LIN {X 0,Y 481.419,Z 1220.363,A -85,B 0,C 180,E1 16137.855,E2 16137.855} C_VEL
LIN {X 0,Y 478.712,Z 1232.005,A -85,B 0,C 180,E1 16135.215,E2 16135.215} C_VEL
LIN {X 0,Y 476.64,Z 1241.797,A -85,B 0,C 180,E1 16132.7,E2 16132.7} C_VEL
LIN {X 0,Y 474.973,Z 1250.804,A -85,B 0,C 180,E1 16130.064,E2 16130.064} C_VEL
LIN {X 0,Y 473.553,Z 1260.287,A -85,B 0,C 180,E1 16126.81,E2 16126.81} C_VEL
LIN {X 0,Y 472.68,Z 1267.551,A -85,B 0,C 180,E1 16123.701,E2 16123.701} C_VEL
LIN {X 0,Y 472.253,Z 1272.478,A -85,B 0,C 180,E1 16121.105,E2 16121.105} C_VEL
LIN {X 0,Y 472.039,Z 1276.348,A -85,B 0,C 180,E1 16118.523,E2 16118.523} C_VEL
LIN {X 0,Y 471.949,Z 1279.075,A -85,B 0,C 180,E1 16116.077,E2 16116.077} C_VEL
LIN {X 0,Y 471.914,Z 1280.879,A -85,B 0,C 180,E1 16113.641,E2 16113.641} C_VEL
LIN {X 0,Y 471.887,Z 1281.781,A -85,B 0,C 180,E1 16111.211,E2 16111.211} C_VEL
LIN {X 0,Y 471.88,Z 1281.802,A -85,B 0,C 180,E1 16108.904,E2 16108.904} C_VEL
LIN {X 0,Y 471.914,Z 1280.943,A -85,B 0,C 180,E1 16106.474,E2 16106.474} C_VEL
LIN {X 0,Y 471.945,Z 1279.181,A -85,B 0,C 180,E1 16104.038,E2 16104.038} C_VEL
LIN {X 0,Y 472.038,Z 1276.338,A -85,B 0,C 180,E1 16101.47,E2 16101.47} C_VEL
LIN {X 0,Y 472.253,Z 1272.465,A -85,B 0,C 180,E1 16098.888,E2 16098.888} C_VEL
LIN {X 0,Y 472.681,Z 1267.536,A -85,B 0,C 180,E1 16096.292,E2 16096.292} C_VEL
LIN {X 0,Y 473.556,Z 1260.267,A -85,B 0,C 180,E1 16093.183,E2 16093.183} C_VEL
LIN {X 0,Y 474.976,Z 1250.78,A -85,B 0,C 180,E1 16089.929,E2 16089.929} C_VEL
LIN {X 0,Y 476.646,Z 1241.775,A -85,B 0,C 180,E1 16087.292,E2 16087.292} C_VEL
LIN {X 0,Y 478.72,Z 1231.982,A -85,B 0,C 180,E1 16084.778,E2 16084.778} C_VEL
LIN {X 0,Y 481.427,Z 1220.335,A -85,B 0,C 180,E1 16082.138,E2 16082.138} C_VEL
LIN {X 0,Y 485.675,Z 1203.701,A -85,B 0,C 180,E1 16078.883,E2 16078.883} C_VEL
LIN {X 0,Y 489.378,Z 1189.815,A -85,B 0,C 180,E1 16076.517,E2 16076.517} C_VEL
LIN {X 0,Y 493.33,Z 1175.667,A -85,B 0,C 180,E1 16074.366,E2 16074.366} C_VEL
LIN {X 0,Y 498.099,Z 1158.939,A -85,B 0,C 180,E1 16072.099,E2 16072.099} C_VEL
LIN {X 0,Y 504.095,Z 1137.823,A -85,B 0,C 180,E1 16069.613,E2 16069.613} C_VEL
LIN {X 0,Y 509.017,Z 1120.127,A -85,B 0,C 180,E1 16067.791,E2 16067.791} C_VEL
LIN {X 0,Y 513.599,Z 1103.252,A -85,B 0,C 180,E1 16066.243,E2 16066.243} C_VEL
LIN {X 0,Y 518.369,Z 1085.032,A -85,B 0,C 180,E1 16064.753,E2 16064.753} C_VEL
LIN {X 0,Y 523.838,Z 1063.175,A -85,B 0,C 180,E1 16063.183,E2 16063.183} C_VEL
LIN {X 0,Y 529.388,Z 1038.821,A -85,B 0,C 180,E1 16061.694,E2 16061.694} C_VEL
LIN {X 0,Y 533.582,Z 1018.565,A -85,B 0,C 180,E1 16060.628,E2 16060.628} C_VEL
LIN {X 0,Y 537.435,Z 998.235,A -85,B 0,C 180,E1 16059.707,E2 16059.707} C_VEL
LIN {X 0,Y 540.948,Z 977.497,A -85,B 0,C 180,E1 16058.905,E2 16058.905} C_VEL
LIN {X 0,Y 544.217,Z 955.344,A -85,B 0,C 180,E1 16058.189,E2 16058.189} C_VEL
LIN {X 0,Y 547.645,Z 926.74,A -85,B 0,C 180,E1 16057.465,E2 16057.465} C_VEL
LIN {X 0,Y 549.736,Z 902.182,A -85,B 0,C 180,E1 16057.006,E2 16057.006} C_VEL
LIN {X 0,Y 559.407,Z 699.055,A -85,B 0,C 180,E1 16053.926,E2 16053.926} C_VEL
LIN {X 0,Y 566.879,Z 547.842,A -85,B 0,C 180,E1 16051.622,E2 16051.622} C_VEL
LIN {X 0,Y 558.19,Z 534.324,A -85,B 0,C 180,E1 16049.808,E2 16049.808} C_VEL
LIN {X 0,Y 548.445,Z 519.702,A -85,B 0,C 180,E1 16047.586,E2 16047.586} C_VEL
LIN {X 0,Y 539.985,Z 507.974,A -85,B 0,C 180,E1 16045.471,E2 16045.471} C_VEL
LIN {X 0,Y 533.469,Z 499.045,A -85,B 0,C 180,E1 16043.677,E2 16043.677} C_VEL
LIN {X 0,Y 530.435,Z 495.224,A -85,B 0,C 180,E1 16042.791,E2 16042.791} C_VEL
LIN {X 0,Y 526.117,Z 489.958,A -85,B 0,C 180,E1 16041.46,E2 16041.46} C_VEL
LIN {X 0,Y 522.215,Z 485.091,A -85,B 0,C 180,E1 16040.16,E2 16040.16} C_VEL
LIN {X 0,Y 517.865,Z 480.177,A -85,B 0,C 180,E1 16038.606,E2 16038.606} C_VEL
LIN {X 0,Y 516.561,Z 478.461,A -85,B 0,C 180,E1 16038.1,E2 16038.1} C_VEL
LIN {X 0,Y 513.201,Z 475.014,A -85,B 0,C 180,E1 16036.76,E2 16036.76} C_VEL
LIN {X 0,Y 511.516,Z 472.461,A -85,B 0,C 180,E1 16035.999,E2 16035.999} C_VEL
LIN {X 0,Y 508.063,Z 469.299,A -85,B 0,C 180,E1 16034.416,E2 16034.416} C_VEL
LIN {X 0,Y 506.144,Z 466.136,A -85,B 0,C 180,E1 16033.364,E2 16033.364} C_VEL
LIN {X 0,Y 502.842,Z 463.782,A -85,B 0,C 180,E1 16031.528,E2 16031.528} C_VEL
LIN {X 0,Y 500.679,Z 459.895,A -85,B 0,C 180,E1 16029.948,E2 16029.948} C_VEL
LIN {X 0,Y 496.132,Z 456.529,A -85,B 0,C 180,E1 16025.9,E2 16025.9} C_VEL
LIN {X 0,Y 494.701,Z 452.911,A -85,B 0,C 180,E1 16023.244,E2 16023.244} C_VEL
LIN {X 0,Y 494.82,Z 453.072,A -85,B 0,C 180,E1 16016.292,E2 16016.292} C_VEL
LIN {X 0,Y 496.254,Z 456.64,A -85,B 0,C 180,E1 16013.754,E2 16013.754} C_VEL
LIN {X 0,Y 500.015,Z 459.457,A -85,B 0,C 180,E1 16010.33,E2 16010.33} C_VEL
LIN {X 0,Y 500.722,Z 459.956,A -85,B 0,C 180,E1 16009.821,E2 16009.821} C_VEL
LIN {X 0,Y 502.632,Z 463.514,A -85,B 0,C 180,E1 16008.409,E2 16008.409} C_VEL
LIN {X 0,Y 505.987,Z 466.072,A -85,B 0,C 180,E1 16006.515,E2 16006.515} C_VEL
LIN {X 0,Y 506.599,Z 466.831,A -85,B 0,C 180,E1 16006.183,E2 16006.183} C_VEL
LIN {X 0,Y 509.251,Z 470.688,A -85,B 0,C 180,E1 16004.804,E2 16004.804} C_VEL
LIN {X 0,Y 512.017,Z 473.051,A -85,B 0,C 180,E1 16003.58,E2 16003.58} C_VEL
LIN {X 0,Y 515.107,Z 477.209,A -85,B 0,C 180,E1 16002.256,E2 16002.256} C_VEL
LIN {X 0,Y 517.415,Z 479.37,A -85,B 0,C 180,E1 16001.377,E2 16001.377} C_VEL
LIN {X 0,Y 520.927,Z 483.776,A -85,B 0,C 180,E1 16000.08,E2 16000.08} C_VEL
LIN {X 0,Y 522.605,Z 485.625,A -85,B 0,C 180,E1 15999.505,E2 15999.505} C_VEL
LIN {X 0,Y 526.557,Z 490.305,A -85,B 0,C 180,E1 15998.208,E2 15998.208} C_VEL
LIN {X 0,Y 532.62,Z 497.875,A -85,B 0,C 180,E1 15996.371,E2 15996.371} C_VEL
LIN {X 0,Y 537.377,Z 503.877,A -85,B 0,C 180,E1 15995.045,E2 15995.045} C_VEL
LIN {X 0,Y 544.823,Z 513.332,A -85,B 0,C 180,E1 15993.132,E2 15993.132} C_VEL
LIN {X 0,Y 555.695,Z 527.944,A -85,B 0,C 180,E1 15990.608,E2 15990.608} C_VEL
LIN {X 0,Y 565.27,Z 542.364,A -85,B 0,C 180,E1 15988.575,E2 15988.575} C_VEL
LIN {X 0,Y 566.874,Z 545.239,A -85,B 0,C 180,E1 15988.242,E2 15988.242} C_VEL
LIN {X 0,Y 556.219,Z 762.388,A -85,B 0,C 180,E1 15984.941,E2 15984.941} C_VEL
LIN {X 0,Y 549.836,Z 895.617,A -85,B 0,C 180,E1 15982.918,E2 15982.918} C_VEL
LIN {X 0,Y 547.564,Z 922.141,A -85,B 0,C 180,E1 15982.412,E2 15982.412} C_VEL
LIN {X 0,Y 544.257,Z 949.115,A -85,B 0,C 180,E1 15981.705,E2 15981.705} C_VEL
LIN {X 0,Y 541.194,Z 970.006,A -85,B 0,C 180,E1 15981.021,E2 15981.021} C_VEL
LIN {X 0,Y 537.814,Z 990.083,A -85,B 0,C 180,E1 15980.241,E2 15980.241} C_VEL
LIN {X 0,Y 533.985,Z 1010.34,A -85,B 0,C 180,E1 15979.322,E2 15979.322} C_VEL
LIN {X 0,Y 529.443,Z 1032.223,A -85,B 0,C 180,E1 15978.164,E2 15978.164} C_VEL
LIN {X 0,Y 523.423,Z 1058.102,A -85,B 0,C 180,E1 15976.546,E2 15976.546} C_VEL
LIN {X 0,Y 518.432,Z 1077.945,A -85,B 0,C 180,E1 15975.098,E2 15975.098} C_VEL
LIN {X 0,Y 513.656,Z 1096.024,A -85,B 0,C 180,E1 15973.602,E2 15973.602} C_VEL
LIN {X 0,Y 508.746,Z 1113.935,A -85,B 0,C 180,E1 15971.933,E2 15971.933} C_VEL
LIN {X 0,Y 502.694,Z 1135.256,A -85,B 0,C 180,E1 15969.667,E2 15969.667} C_VEL
LIN {X 0,Y 499.787,Z 1145.411,A -85,B 0,C 180,E1 15968.454,E2 15968.454} C_VEL
LIN {X 0,Y 497.444,Z 1150.756,A -85,B 0,C 180,E1 15967.865,E2 15967.865} C_VEL
LIN {X 0,Y 488.416,Z 1164.255,A -85,B 0,C 180,E1 15966.475,E2 15966.475} C_VEL
LIN {X 0,Y 486.11,Z 1169.146,A -85,B 0,C 180,E1 15965.825,E2 15965.825} C_VEL
LIN {X 0,Y 481.158,Z 1186.125,A -85,B 0,C 180,E1 15963.126,E2 15963.126} C_VEL
LIN {X 0,Y 476.645,Z 1201.723,A -85,B 0,C 180,E1 15960.232,E2 15960.232} C_VEL
LIN {X 0,Y 473.56,Z 1213.335,A -85,B 0,C 180,E1 15957.786,E2 15957.786} C_VEL
LIN {X 0,Y 470.892,Z 1224.082,A -85,B 0,C 180,E1 15955.234,E2 15955.234} C_VEL
LIN {X 0,Y 468.337,Z 1235.729,A -85,B 0,C 180,E1 15952.074,E2 15952.074} C_VEL
LIN {X 0,Y 466.403,Z 1245.831,A -85,B 0,C 180,E1 15948.761,E2 15948.761} C_VEL
LIN {X 0,Y 465.348,Z 1252.735,A -85,B 0,C 180,E1 15946.095,E2 15946.095} C_VEL
LIN {X 0,Y 464.648,Z 1258.556,A -85,B 0,C 180,E1 15943.424,E2 15943.424} C_VEL
LIN {X 0,Y 464.225,Z 1263.433,A -85,B 0,C 180,E1 15940.678,E2 15940.678} C_VEL
LIN {X 0,Y 463.98,Z 1268,A -85,B 0,C 180,E1 15937.308,E2 15937.308} C_VEL
LIN {X 0,Y 463.917,Z 1270.577,A -85,B 0,C 180,E1 15934.206,E2 15934.206} C_VEL
LIN {X 0,Y 463.905,Z 1271.703,A -85,B 0,C 180,E1 15931.609,E2 15931.609} C_VEL
LIN {X 0,Y 463.872,Z 1271.834,A -85,B 0,C 180,E1 15929.016,E2 15929.016} C_VEL
LIN {X 0,Y 463.912,Z 1271.04,A -85,B 0,C 180,E1 15926.544,E2 15926.544} C_VEL
LIN {X 0,Y 463.95,Z 1269.227,A -85,B 0,C 180,E1 15923.942,E2 15923.942} C_VEL
LIN {X 0,Y 464.049,Z 1266.403,A -85,B 0,C 180,E1 15921.329,E2 15921.329} C_VEL
LIN {X 0,Y 464.286,Z 1262.364,A -85,B 0,C 180,E1 15918.576,E2 15918.576} C_VEL
LIN {X 0,Y 464.772,Z 1257.203,A -85,B 0,C 180,E1 15915.808,E2 15915.808} C_VEL
LIN {X 0,Y 465.874,Z 1249.153,A -85,B 0,C 180,E1 15912.354,E2 15912.354} C_VEL
LIN {X 0,Y 467.362,Z 1240.467,A -85,B 0,C 180,E1 15909.334,E2 15909.334} C_VEL
LIN {X 0,Y 469.114,Z 1231.79,A -85,B 0,C 180,E1 15906.73,E2 15906.73} C_VEL
LIN {X 0,Y 471.317,Z 1222.278,A -85,B 0,C 180,E1 15904.226,E2 15904.226} C_VEL
LIN {X 0,Y 474.554,Z 1209.618,A -85,B 0,C 180,E1 15901.294,E2 15901.294} C_VEL
LIN {X 0,Y 478.758,Z 1194.258,A -85,B 0,C 180,E1 15898.25,E2 15898.25} C_VEL
LIN {X 0,Y 482.501,Z 1181.259,A -85,B 0,C 180,E1 15895.983,E2 15895.983} C_VEL
LIN {X 0,Y 486.555,Z 1167.656,A -85,B 0,C 180,E1 15893.864,E2 15893.864} C_VEL
LIN {X 0,Y 491.218,Z 1152.193,A -85,B 0,C 180,E1 15891.711,E2 15891.711} C_VEL
LIN {X 0,Y 497.188,Z 1132.548,A -85,B 0,C 180,E1 15889.304,E2 15889.304} C_VEL
LIN {X 0,Y 502.899,Z 1113.013,A -85,B 0,C 180,E1 15887.242,E2 15887.242} C_VEL
LIN {X 0,Y 507.858,Z 1095.621,A -85,B 0,C 180,E1 15885.618,E2 15885.618} C_VEL
LIN {X 0,Y 512.717,Z 1077.884,A -85,B 0,C 180,E1 15884.145,E2 15884.145} C_VEL
LIN {X 0,Y 517.775,Z 1058.428,A -85,B 0,C 180,E1 15882.718,E2 15882.718} C_VEL
LIN {X 0,Y 523.999,Z 1032.581,A -85,B 0,C 180,E1 15881.093,E2 15881.093} C_VEL
LIN {X 0,Y 528.687,Z 1010.722,A -85,B 0,C 180,E1 15879.931,E2 15879.931} C_VEL
LIN {X 0,Y 532.643,Z 990.44,A -85,B 0,C 180,E1 15879.006,E2 15879.006} C_VEL
LIN {X 0,Y 536.242,Z 969.723,A -85,B 0,C 180,E1 15878.201,E2 15878.201} C_VEL
LIN {X 0,Y 539.707,Z 946.697,A -85,B 0,C 180,E1 15877.455,E2 15877.455} C_VEL
LIN {X 0,Y 543.153,Z 917.776,A -85,B 0,C 180,E1 15876.73,E2 15876.73} C_VEL
LIN {X 0,Y 545.156,Z 894.477,A -85,B 0,C 180,E1 15876.295,E2 15876.295} C_VEL
LIN {X 0,Y 555.378,Z 688.317,A -85,B 0,C 180,E1 15873.155,E2 15873.155} C_VEL
LIN {X 0,Y 562.529,Z 549.365,A -85,B 0,C 180,E1 15871.029,E2 15871.029} C_VEL
LIN {X 0,Y 552.764,Z 534.378,A -85,B 0,C 180,E1 15868.907,E2 15868.907} C_VEL
LIN {X 0,Y 541.403,Z 519.012,A -85,B 0,C 180,E1 15866.193,E2 15866.193} C_VEL
LIN {X 0,Y 532.717,Z 507.898,A -85,B 0,C 180,E1 15863.859,E2 15863.859} C_VEL
LIN {X 0,Y 528.301,Z 502.407,A -85,B 0,C 180,E1 15862.559,E2 15862.559} C_VEL
LIN {X 0,Y 524.158,Z 497.301,A -85,B 0,C 180,E1 15861.251,E2 15861.251} C_VEL
LIN {X 0,Y 519.573,Z 491.687,A -85,B 0,C 180,E1 15859.681,E2 15859.681} C_VEL
LIN {X 0,Y 515.874,Z 487.212,A -85,B 0,C 180,E1 15858.3,E2 15858.3} C_VEL
LIN {X 0,Y 514.503,Z 485.734,A -85,B 0,C 180,E1 15857.765,E2 15857.765} C_VEL
LIN {X 0,Y 511.154,Z 481.865,A -85,B 0,C 180,E1 15856.361,E2 15856.361} C_VEL
LIN {X 0,Y 509.976,Z 480.144,A -85,B 0,C 180,E1 15855.815,E2 15855.815} C_VEL
LIN {X 0,Y 506.51,Z 476.774,A -85,B 0,C 180,E1 15854.169,E2 15854.169} C_VEL
LIN {X 0,Y 504.733,Z 473.91,A -85,B 0,C 180,E1 15853.169,E2 15853.169} C_VEL
LIN {X 0,Y 501.451,Z 471.401,A -85,B 0,C 180,E1 15851.269,E2 15851.269} C_VEL
LIN {X 0,Y 499.227,Z 467.473,A -85,B 0,C 180,E1 15849.569,E2 15849.569} C_VEL
LIN {X 0,Y 495.28,Z 464.726,A -85,B 0,C 180,E1 15845.91,E2 15845.91} C_VEL
LIN {X 0,Y 493.731,Z 460.864,A -85,B 0,C 180,E1 15842.786,E2 15842.786} C_VEL
LIN {X 0,Y 493.807,Z 461.029,A -85,B 0,C 180,E1 15837.098,E2 15837.098} C_VEL
LIN {X 0,Y 495.742,Z 465.272,A -85,B 0,C 180,E1 15833.631,E2 15833.631} C_VEL
LIN {X 0,Y 499.508,Z 467.827,A -85,B 0,C 180,E1 15830.32,E2 15830.32} C_VEL
LIN {X 0,Y 501.609,Z 471.614,A -85,B 0,C 180,E1 15828.735,E2 15828.735} C_VEL
LIN {X 0,Y 505.115,Z 474.417,A -85,B 0,C 180,E1 15826.725,E2 15826.725} C_VEL
LIN {X 0,Y 508.144,Z 478.707,A -85,B 0,C 180,E1 15825.12,E2 15825.12} C_VEL
LIN {X 0,Y 510.497,Z 480.794,A -85,B 0,C 180,E1 15824.056,E2 15824.056} C_VEL
LIN {X 0,Y 513.661,Z 485.023,A -85,B 0,C 180,E1 15822.673,E2 15822.673} C_VEL
LIN {X 0,Y 515.722,Z 486.993,A -85,B 0,C 180,E1 15821.87,E2 15821.87} C_VEL
LIN {X 0,Y 519.4,Z 491.534,A -85,B 0,C 180,E1 15820.488,E2 15820.488} C_VEL
LIN {X 0,Y 521.036,Z 493.538,A -85,B 0,C 180,E1 15819.909,E2 15819.909} C_VEL
LIN {X 0,Y 525.9,Z 499.458,A -85,B 0,C 180,E1 15818.297,E2 15818.297} C_VEL
LIN {X 0,Y 530.608,Z 505.302,A -85,B 0,C 180,E1 15816.859,E2 15816.859} C_VEL
LIN {X 0,Y 536.955,Z 514.063,A -85,B 0,C 180,E1 15815.053,E2 15815.053} C_VEL
LIN {X 0,Y 543.856,Z 523.758,A -85,B 0,C 180,E1 15813.258,E2 15813.258} C_VEL
LIN {X 0,Y 552.297,Z 536.23,A -85,B 0,C 180,E1 15811.241,E2 15811.241} C_VEL
LIN {X 0,Y 562.019,Z 551.359,A -85,B 0,C 180,E1 15809.118,E2 15809.118} C_VEL
LIN {X 0,Y 562.519,Z 552.506,A -85,B 0,C 180,E1 15809.005,E2 15809.005} C_VEL
LIN {X 0,Y 551.538,Z 769.195,A -85,B 0,C 180,E1 15805.698,E2 15805.698} C_VEL
LIN {X 0,Y 544.926,Z 902.792,A -85,B 0,C 180,E1 15803.66,E2 15803.66} C_VEL
LIN {X 0,Y 542.526,Z 929.769,A -85,B 0,C 180,E1 15803.148,E2 15803.148} C_VEL
LIN {X 0,Y 539.082,Z 956.677,A -85,B 0,C 180,E1 15802.446,E2 15802.446} C_VEL
LIN {X 0,Y 535.875,Z 977.691,A -85,B 0,C 180,E1 15801.762,E2 15801.762} C_VEL
LIN {X 0,Y 532.498,Z 997.1,A -85,B 0,C 180,E1 15801.013,E2 15801.013} C_VEL
LIN {X 0,Y 528.51,Z 1017.543,A -85,B 0,C 180,E1 15800.092,E2 15800.092} C_VEL
LIN {X 0,Y 524.246,Z 1037.558,A -85,B 0,C 180,E1 15799.042,E2 15799.042} C_VEL
LIN {X 0,Y 518.513,Z 1062.103,A -85,B 0,C 180,E1 15797.551,E2 15797.551} C_VEL
LIN {X 0,Y 512.9,Z 1083.81,A -85,B 0,C 180,E1 15795.994,E2 15795.994} C_VEL
LIN {X 0,Y 508.189,Z 1101.184,A -85,B 0,C 180,E1 15794.581,E2 15794.581} C_VEL
LIN {X 0,Y 503.406,Z 1118.141,A -85,B 0,C 180,E1 15793.034,E2 15793.034} C_VEL
LIN {X 0,Y 498.461,Z 1135.191,A -85,B 0,C 180,E1 15791.29,E2 15791.29} C_VEL
LIN {X 0,Y 493.227,Z 1153.063,A -85,B 0,C 180,E1 15789.228,E2 15789.228} C_VEL
LIN {X 0,Y 487.168,Z 1173.445,A -85,B 0,C 180,E1 15786.521,E2 15786.521} C_VEL
LIN {X 0,Y 482.821,Z 1188.219,A -85,B 0,C 180,E1 15784.278,E2 15784.278} C_VEL
LIN {X 0,Y 479.025,Z 1201.533,A -85,B 0,C 180,E1 15782.012,E2 15782.012} C_VEL
LIN {X 0,Y 475.415,Z 1214.893,A -85,B 0,C 180,E1 15779.457,E2 15779.457} C_VEL
LIN {X 0,Y 471.628,Z 1229.839,A -85,B 0,C 180,E1 15776.161,E2 15776.161} C_VEL
LIN {X 0,Y 469.247,Z 1240.319,A -85,B 0,C 180,E1 15773.477,E2 15773.477} C_VEL
LIN {X 0,Y 467.508,Z 1249.081,A -85,B 0,C 180,E1 15770.922,E2 15770.922} C_VEL
LIN {X 0,Y 466.111,Z 1257.063,A -85,B 0,C 180,E1 15768.247,E2 15768.247} C_VEL
LIN {X 0,Y 465.127,Z 1264.171,A -85,B 0,C 180,E1 15765.455,E2 15765.455} C_VEL
LIN {X 0,Y 464.372,Z 1271.415,A -85,B 0,C 180,E1 15761.925,E2 15761.925} C_VEL
LIN {X 0,Y 464.051,Z 1275.866,A -85,B 0,C 180,E1 15759.046,E2 15759.046} C_VEL
LIN {X 0,Y 463.959,Z 1278.845,A -85,B 0,C 180,E1 15756.431,E2 15756.431} C_VEL
LIN {X 0,Y 463.916,Z 1280.743,A -85,B 0,C 180,E1 15753.951,E2 15753.951} C_VEL
LIN {X 0,Y 463.902,Z 1281.735,A -85,B 0,C 180,E1 15751.478,E2 15751.478} C_VEL
LIN {X 0,Y 463.875,Z 1281.824,A -85,B 0,C 180,E1 15749.008,E2 15749.008} C_VEL
LIN {X 0,Y 463.914,Z 1281.011,A -85,B 0,C 180,E1 15746.537,E2 15746.537} C_VEL
LIN {X 0,Y 463.949,Z 1279.178,A -85,B 0,C 180,E1 15743.935,E2 15743.935} C_VEL
LIN {X 0,Y 464.05,Z 1276.335,A -85,B 0,C 180,E1 15741.322,E2 15741.322} C_VEL
LIN {X 0,Y 464.265,Z 1272.654,A -85,B 0,C 180,E1 15738.82,E2 15738.82} C_VEL
LIN {X 0,Y 464.706,Z 1267.729,A -85,B 0,C 180,E1 15736.179,E2 15736.179} C_VEL
LIN {X 0,Y 465.528,Z 1261.094,A -85,B 0,C 180,E1 15733.27,E2 15733.27} C_VEL
LIN {X 0,Y 467.047,Z 1251.505,A -85,B 0,C 180,E1 15729.835,E2 15729.835} C_VEL
LIN {X 0,Y 468.861,Z 1242.145,A -85,B 0,C 180,E1 15727.026,E2 15727.026} C_VEL
LIN {X 0,Y 471.035,Z 1232.409,A -85,B 0,C 180,E1 15724.472,E2 15724.472} C_VEL
LIN {X 0,Y 473.711,Z 1221.398,A -85,B 0,C 180,E1 15721.918,E2 15721.918} C_VEL
LIN {X 0,Y 477.562,Z 1207.101,A -85,B 0,C 180,E1 15718.996,E2 15718.996} C_VEL
LIN {X 0,Y 481.936,Z 1191.272,A -85,B 0,C 180,E1 15716.216,E2 15716.216} C_VEL
LIN {X 0,Y 486.155,Z 1176.791,A -85,B 0,C 180,E1 15713.967,E2 15713.967} C_VEL
LIN {X 0,Y 490.64,Z 1161.636,A -85,B 0,C 180,E1 15711.865,E2 15711.865} C_VEL
LIN {X 0,Y 496.05,Z 1143.538,A -85,B 0,C 180,E1 15709.636,E2 15709.636} C_VEL
LIN {X 0,Y 502.349,Z 1121.865,A -85,B 0,C 180,E1 15707.331,E2 15707.331} C_VEL
LIN {X 0,Y 507.37,Z 1104.081,A -85,B 0,C 180,E1 15705.674,E2 15705.674} C_VEL
LIN {X 0,Y 512.117,Z 1086.627,A -85,B 0,C 180,E1 15704.228,E2 15704.228} C_VEL
LIN {X 0,Y 516.949,Z 1067.962,A -85,B 0,C 180,E1 15702.854,E2 15702.854} C_VEL
LIN {X 0,Y 522.724,Z 1044.339,A -85,B 0,C 180,E1 15701.339,E2 15701.339} C_VEL
LIN {X 0,Y 528.073,Z 1019.603,A -85,B 0,C 180,E1 15700.011,E2 15700.011} C_VEL
LIN {X 0,Y 532.037,Z 999.427,A -85,B 0,C 180,E1 15699.087,E2 15699.087} C_VEL
LIN {X 0,Y 535.649,Z 978.884,A -85,B 0,C 180,E1 15698.283,E2 15698.283} C_VEL
LIN {X 0,Y 538.892,Z 957.744,A -85,B 0,C 180,E1 15697.589,E2 15697.589} C_VEL
LIN {X 0,Y 542.016,Z 933.624,A -85,B 0,C 180,E1 15696.946,E2 15696.946} C_VEL
LIN {X 0,Y 544.766,Z 904.653,A -85,B 0,C 180,E1 15696.373,E2 15696.373} C_VEL
LIN {X 0,Y 548.192,Z 837.513,A -85,B 0,C 180,E1 15695.34,E2 15695.34} C_VEL
LIN {X 0,Y 558.918,Z 620.585,A -85,B 0,C 180,E1 15692.04,E2 15692.04} C_VEL
LIN {X 0,Y 562.397,Z 552.084,A -85,B 0,C 180,E1 15690.978,E2 15690.978} C_VEL
LIN {X 0,Y 553.476,Z 538.084,A -85,B 0,C 180,E1 15689.046,E2 15689.046} C_VEL
LIN {X 0,Y 544.949,Z 525.376,A -85,B 0,C 180,E1 15687.038,E2 15687.038} C_VEL
LIN {X 0,Y 537.505,Z 514.862,A -85,B 0,C 180,E1 15685.126,E2 15685.126} C_VEL
LIN {X 0,Y 530.745,Z 505.498,A -85,B 0,C 180,E1 15683.217,E2 15683.217} C_VEL
LIN {X 0,Y 527.928,Z 502.032,A -85,B 0,C 180,E1 15682.377,E2 15682.377} C_VEL
LIN {X 0,Y 524.176,Z 497.346,A -85,B 0,C 180,E1 15681.191,E2 15681.191} C_VEL
LIN {X 0,Y 519.572,Z 491.7,A -85,B 0,C 180,E1 15679.622,E2 15679.622} C_VEL
LIN {X 0,Y 515.853,Z 487.221,A -85,B 0,C 180,E1 15678.243,E2 15678.243} C_VEL
LIN {X 0,Y 514.617,Z 485.836,A -85,B 0,C 180,E1 15677.761,E2 15677.761} C_VEL
LIN {X 0,Y 511.231,Z 482.013,A -85,B 0,C 180,E1 15676.358,E2 15676.358} C_VEL
LIN {X 0,Y 510.053,Z 480.185,A -85,B 0,C 180,E1 15675.813,E2 15675.813} C_VEL
LIN {X 0,Y 506.544,Z 476.847,A -85,B 0,C 180,E1 15674.168,E2 15674.168} C_VEL
LIN {X 0,Y 504.751,Z 473.922,A -85,B 0,C 180,E1 15673.168,E2 15673.168} C_VEL
LIN {X 0,Y 501.431,Z 471.371,A -85,B 0,C 180,E1 15671.269,E2 15671.269} C_VEL
LIN {X 0,Y 499.167,Z 467.442,A -85,B 0,C 180,E1 15669.57,E2 15669.57} C_VEL
LIN {X 0,Y 495.337,Z 464.784,A -85,B 0,C 180,E1 15666.142,E2 15666.142} C_VEL
LIN {X 0,Y 493.671,Z 460.844,A -85,B 0,C 180,E1 15663.135,E2 15663.135} C_VEL
LIN {X 0,Y 493.79,Z 460.974,A -85,B 0,C 180,E1 15656.401,E2 15656.401} C_VEL
LIN {X 0,Y 495.186,Z 464.519,A -85,B 0,C 180,E1 15653.856,E2 15653.856} C_VEL
LIN {X 0,Y 498.894,Z 467.351,A -85,B 0,C 180,E1 15650.424,E2 15650.424} C_VEL
LIN {X 0,Y 499.505,Z 467.867,A -85,B 0,C 180,E1 15649.971,E2 15649.971} C_VEL
LIN {X 0,Y 501.483,Z 471.417,A -85,B 0,C 180,E1 15648.499,E2 15648.499} C_VEL
LIN {X 0,Y 505.11,Z 474.388,A -85,B 0,C 180,E1 15646.433,E2 15646.433} C_VEL
LIN {X 0,Y 507.821,Z 478.379,A -85,B 0,C 180,E1 15644.994,E2 15644.994} C_VEL
LIN {X 0,Y 510.484,Z 480.731,A -85,B 0,C 180,E1 15643.792,E2 15643.792} C_VEL
LIN {X 0,Y 513.739,Z 485.029,A -85,B 0,C 180,E1 15642.383,E2 15642.383} C_VEL
LIN {X 0,Y 515.742,Z 486.957,A -85,B 0,C 180,E1 15641.607,E2 15641.607} C_VEL
LIN {X 0,Y 519.364,Z 491.466,A -85,B 0,C 180,E1 15640.252,E2 15640.252} C_VEL
LIN {X 0,Y 521.084,Z 493.559,A -85,B 0,C 180,E1 15639.647,E2 15639.647} C_VEL
LIN {X 0,Y 525.893,Z 499.386,A -85,B 0,C 180,E1 15638.061,E2 15638.061} C_VEL
LIN {X 0,Y 530.597,Z 505.253,A -85,B 0,C 180,E1 15636.629,E2 15636.629} C_VEL
LIN {X 0,Y 535.39,Z 511.381,A -85,B 0,C 180,E1 15635.27,E2 15635.27} C_VEL
LIN {X 0,Y 542.663,Z 520.763,A -85,B 0,C 180,E1 15633.371,E2 15633.371} C_VEL
LIN {X 0,Y 553.115,Z 534.981,A -85,B 0,C 180,E1 15630.903,E2 15630.903} C_VEL
LIN {X 0,Y 562.472,Z 549.3,A -85,B 0,C 180,E1 15628.878,E2 15628.878} C_VEL
LIN {X 0,Y 551.643,Z 762.631,A -85,B 0,C 180,E1 15625.621,E2 15625.621} C_VEL
LIN {X 0,Y 545.038,Z 895.729,A -85,B 0,C 180,E1 15623.591,E2 15623.591} C_VEL
LIN {X 0,Y 542.693,Z 922.339,A -85,B 0,C 180,E1 15623.082,E2 15623.082} C_VEL
LIN {X 0,Y 539.287,Z 949.325,A -85,B 0,C 180,E1 15622.373,E2 15622.373} C_VEL
LIN {X 0,Y 536.026,Z 970.844,A -85,B 0,C 180,E1 15621.666,E2 15621.666} C_VEL
LIN {X 0,Y 532.442,Z 991.404,A -85,B 0,C 180,E1 15620.86,E2 15620.86} C_VEL
LIN {X 0,Y 528.266,Z 1012.692,A -85,B 0,C 180,E1 15619.88,E2 15619.88} C_VEL
LIN {X 0,Y 522.486,Z 1038.981,A -85,B 0,C 180,E1 15618.442,E2 15618.442} C_VEL
LIN {X 0,Y 517.18,Z 1060.623,A -85,B 0,C 180,E1 15617.037,E2 15617.037} C_VEL
LIN {X 0,Y 512.443,Z 1078.806,A -85,B 0,C 180,E1 15615.69,E2 15615.69} C_VEL
LIN {X 0,Y 507.598,Z 1096.478,A -85,B 0,C 180,E1 15614.215,E2 15614.215} C_VEL
LIN {X 0,Y 502.258,Z 1115.242,A -85,B 0,C 180,E1 15612.447,E2 15612.447} C_VEL
LIN {X 0,Y 495.703,Z 1137.269,A -85,B 0,C 180,E1 15610.052,E2 15610.052} C_VEL
LIN {X 0,Y 490.707,Z 1153.829,A -85,B 0,C 180,E1 15607.981,E2 15607.981} C_VEL
LIN {X 0,Y 486.216,Z 1168.784,A -85,B 0,C 180,E1 15605.879,E2 15605.879} C_VEL
LIN {X 0,Y 486.11,Z 1169.146,A -85,B 0,C 180,E1 15605.825,E2 15605.825} C_VEL
LIN {X 0,Y 483.843,Z 1174.1,A -85,B 0,C 180,E1 15605.162,E2 15605.162} C_VEL
LIN {X 0,Y 474.567,Z 1187.024,A -85,B 0,C 180,E1 15603.482,E2 15603.482} C_VEL
LIN {X 0,Y 472.731,Z 1190.74,A -85,B 0,C 180,E1 15602.858,E2 15602.858} C_VEL
LIN {X 0,Y 469.054,Z 1203.08,A -85,B 0,C 180,E1 15600.49,E2 15600.49} C_VEL
LIN {X 0,Y 465.9,Z 1214.435,A -85,B 0,C 180,E1 15598.037,E2 15598.037} C_VEL
LIN {X 0,Y 462.783,Z 1226.606,A -85,B 0,C 180,E1 15595.057,E2 15595.057} C_VEL
LIN {X 0,Y 460.106,Z 1238.252,A -85,B 0,C 180,E1 15591.684,E2 15591.684} C_VEL
LIN {X 0,Y 458.525,Z 1246.273,A -85,B 0,C 180,E1 15588.963,E2 15588.963} C_VEL
LIN {X 0,Y 457.415,Z 1253.127,A -85,B 0,C 180,E1 15586.251,E2 15586.251} C_VEL
LIN {X 0,Y 456.686,Z 1258.863,A -85,B 0,C 180,E1 15583.552,E2 15583.552} C_VEL
LIN {X 0,Y 456.223,Z 1263.932,A -85,B 0,C 180,E1 15580.612,E2 15580.612} C_VEL
LIN {X 0,Y 455.984,Z 1268.279,A -85,B 0,C 180,E1 15577.184,E2 15577.184} C_VEL
LIN {X 0,Y 455.917,Z 1270.672,A -85,B 0,C 180,E1 15574.154,E2 15574.154} C_VEL
LIN {X 0,Y 455.904,Z 1271.741,A -85,B 0,C 180,E1 15571.512,E2 15571.512} C_VEL
LIN {X 0,Y 455.873,Z 1271.848,A -85,B 0,C 180,E1 15568.998,E2 15568.998} C_VEL
LIN {X 0,Y 455.912,Z 1271.062,A -85,B 0,C 180,E1 15566.483,E2 15566.483} C_VEL
LIN {X 0,Y 455.953,Z 1269.266,A -85,B 0,C 180,E1 15563.835,E2 15563.835} C_VEL
LIN {X 0,Y 456.057,Z 1266.471,A -85,B 0,C 180,E1 15561.176,E2 15561.176} C_VEL
LIN {X 0,Y 456.304,Z 1262.656,A -85,B 0,C 180,E1 15558.502,E2 15558.502} C_VEL
LIN {X 0,Y 456.785,Z 1257.794,A -85,B 0,C 180,E1 15555.813,E2 15555.813} C_VEL
LIN {X 0,Y 457.759,Z 1250.951,A -85,B 0,C 180,E1 15552.723,E2 15552.723} C_VEL
LIN {X 0,Y 459.457,Z 1241.359,A -85,B 0,C 180,E1 15549.228,E2 15549.228} C_VEL
LIN {X 0,Y 461.371,Z 1232.339,A -85,B 0,C 180,E1 15546.454,E2 15546.454} C_VEL
LIN {X 0,Y 463.672,Z 1222.877,A -85,B 0,C 180,E1 15543.907,E2 15543.907} C_VEL
LIN {X 0,Y 466.722,Z 1211.414,A -85,B 0,C 180,E1 15541.187,E2 15541.187} C_VEL
LIN {X 0,Y 471.246,Z 1195.738,A -85,B 0,C 180,E1 15537.97,E2 15537.97} C_VEL
LIN {X 0,Y 475.577,Z 1181.347,A -85,B 0,C 180,E1 15535.418,E2 15535.418} C_VEL
LIN {X 0,Y 479.817,Z 1167.744,A -85,B 0,C 180,E1 15533.274,E2 15533.274} C_VEL
LIN {X 0,Y 484.702,Z 1152.233,A -85,B 0,C 180,E1 15531.093,E2 15531.093} C_VEL
LIN {X 0,Y 490.977,Z 1132.377,A -85,B 0,C 180,E1 15528.642,E2 15528.642} C_VEL
LIN {X 0,Y 496.805,Z 1113.177,A -85,B 0,C 180,E1 15526.599,E2 15526.599} C_VEL
LIN {X 0,Y 501.86,Z 1096.108,A -85,B 0,C 180,E1 15524.993,E2 15524.993} C_VEL
LIN {X 0,Y 506.92,Z 1078.302,A -85,B 0,C 180,E1 15523.504,E2 15523.504} C_VEL
LIN {X 0,Y 512.025,Z 1059.321,A -85,B 0,C 180,E1 15522.1,E2 15522.1} C_VEL
LIN {X 0,Y 518.219,Z 1034.667,A -85,B 0,C 180,E1 15520.525,E2 15520.525} C_VEL
LIN {X 0,Y 523.267,Z 1011.93,A -85,B 0,C 180,E1 15519.303,E2 15519.303} C_VEL
LIN {X 0,Y 527.335,Z 991.802,A -85,B 0,C 180,E1 15518.376,E2 15518.376} C_VEL
LIN {X 0,Y 531.032,Z 971.278,A -85,B 0,C 180,E1 15517.569,E2 15517.569} C_VEL
LIN {X 0,Y 534.371,Z 949.913,A -85,B 0,C 180,E1 15516.864,E2 15516.864} C_VEL
LIN {X 0,Y 537.853,Z 923.349,A -85,B 0,C 180,E1 15516.16,E2 15516.16} C_VEL
LIN {X 0,Y 540.341,Z 896.071,A -85,B 0,C 180,E1 15515.635,E2 15515.635} C_VEL
LIN {X 0,Y 546.277,Z 780.939,A -85,B 0,C 180,E1 15513.868,E2 15513.868} C_VEL
LIN {X 0,Y 557.775,Z 561.683,A -85,B 0,C 180,E1 15510.514,E2 15510.514} C_VEL
LIN {X 0,Y 558.119,Z 553.711,A -85,B 0,C 180,E1 15510.375,E2 15510.375} C_VEL
LIN {X 0,Y 549.798,Z 540.875,A -85,B 0,C 180,E1 15508.516,E2 15508.516} C_VEL
LIN {X 0,Y 539.081,Z 526.157,A -85,B 0,C 180,E1 15505.9,E2 15505.9} C_VEL
LIN {X 0,Y 530.508,Z 515.057,A -85,B 0,C 180,E1 15503.552,E2 15503.552} C_VEL
LIN {X 0,Y 526.259,Z 509.699,A -85,B 0,C 180,E1 15502.275,E2 15502.275} C_VEL
LIN {X 0,Y 522.235,Z 504.686,A -85,B 0,C 180,E1 15500.98,E2 15500.98} C_VEL
LIN {X 0,Y 517.714,Z 499.101,A -85,B 0,C 180,E1 15499.402,E2 15499.402} C_VEL
LIN {X 0,Y 513.966,Z 494.383,A -85,B 0,C 180,E1 15497.966,E2 15497.966} C_VEL
LIN {X 0,Y 509.802,Z 489.784,A -85,B 0,C 180,E1 15496.23,E2 15496.23} C_VEL
LIN {X 0,Y 508.524,Z 487.863,A -85,B 0,C 180,E1 15495.627,E2 15495.627} C_VEL
LIN {X 0,Y 505.006,Z 484.321,A -85,B 0,C 180,E1 15493.92,E2 15493.92} C_VEL
LIN {X 0,Y 503.352,Z 481.691,A -85,B 0,C 180,E1 15492.972,E2 15492.972} C_VEL
LIN {X 0,Y 500.057,Z 478.988,A -85,B 0,C 180,E1 15491.009,E2 15491.009} C_VEL
LIN {X 0,Y 498.106,Z 475.368,A -85,B 0,C 180,E1 15489.474,E2 15489.474} C_VEL
LIN {X 0,Y 494.217,Z 472.605,A -85,B 0,C 180,E1 15485.806,E2 15485.806} C_VEL
LIN {X 0,Y 492.711,Z 468.8,A -85,B 0,C 180,E1 15482.675,E2 15482.675} C_VEL
LIN {X 0,Y 492.788,Z 468.926,A -85,B 0,C 180,E1 15477.209,E2 15477.209} C_VEL
LIN {X 0,Y 494.768,Z 473.249,A -85,B 0,C 180,E1 15473.618,E2 15473.618} C_VEL
LIN {X 0,Y 498.303,Z 475.703,A -85,B 0,C 180,E1 15470.471,E2 15470.471} C_VEL
LIN {X 0,Y 500.462,Z 479.513,A -85,B 0,C 180,E1 15468.825,E2 15468.825} C_VEL
LIN {X 0,Y 503.732,Z 482.154,A -85,B 0,C 180,E1 15466.921,E2 15466.921} C_VEL
LIN {X 0,Y 506.833,Z 486.511,A -85,B 0,C 180,E1 15465.256,E2 15465.256} C_VEL
LIN {X 0,Y 508.975,Z 488.466,A -85,B 0,C 180,E1 15464.27,E2 15464.27} C_VEL
LIN {X 0,Y 512.166,Z 492.711,A -85,B 0,C 180,E1 15462.855,E2 15462.855} C_VEL
LIN {X 0,Y 514.126,Z 494.675,A -85,B 0,C 180,E1 15462.075,E2 15462.075} C_VEL
LIN {X 0,Y 517.993,Z 499.359,A -85,B 0,C 180,E1 15460.609,E2 15460.609} C_VEL
LIN {X 0,Y 524.11,Z 507.052,A -85,B 0,C 180,E1 15458.513,E2 15458.513} C_VEL
LIN {X 0,Y 528.667,Z 512.77,A -85,B 0,C 180,E1 15457.099,E2 15457.099} C_VEL
LIN {X 0,Y 534.959,Z 521.593,A -85,B 0,C 180,E1 15455.278,E2 15455.278} C_VEL
LIN {X 0,Y 543.547,Z 533.805,A -85,B 0,C 180,E1 15453.034,E2 15453.034} C_VEL
LIN {X 0,Y 553.888,Z 549.763,A -85,B 0,C 180,E1 15450.592,E2 15450.592} C_VEL
LIN {X 0,Y 558.175,Z 556.88,A -85,B 0,C 180,E1 15449.645,E2 15449.645} C_VEL
LIN {X 0,Y 546.865,Z 772.7,A -85,B 0,C 180,E1 15446.34,E2 15446.34} C_VEL
LIN {X 0,Y 540.203,Z 902.723,A -85,B 0,C 180,E1 15444.347,E2 15444.347} C_VEL
LIN {X 0,Y 537.723,Z 929.853,A -85,B 0,C 180,E1 15443.83,E2 15443.83} C_VEL
LIN {X 0,Y 534.217,Z 956.489,A -85,B 0,C 180,E1 15443.135,E2 15443.135} C_VEL
LIN {X 0,Y 530.896,Z 977.61,A -85,B 0,C 180,E1 15442.45,E2 15442.45} C_VEL
LIN {X 0,Y 527.176,Z 998.303,A -85,B 0,C 180,E1 15441.646,E2 15441.646} C_VEL
LIN {X 0,Y 523.074,Z 1018.593,A -85,B 0,C 180,E1 15440.723,E2 15440.723} C_VEL
LIN {X 0,Y 517.785,Z 1042.51,A -85,B 0,C 180,E1 15439.446,E2 15439.446} C_VEL
LIN {X 0,Y 511.776,Z 1066.482,A -85,B 0,C 180,E1 15437.922,E2 15437.922} C_VEL
LIN {X 0,Y 506.772,Z 1085.197,A -85,B 0,C 180,E1 15436.551,E2 15436.551} C_VEL
LIN {X 0,Y 501.803,Z 1102.828,A -85,B 0,C 180,E1 15435.095,E2 15435.095} C_VEL
LIN {X 0,Y 496.754,Z 1120.04,A -85,B 0,C 180,E1 15433.496,E2 15433.496} C_VEL
LIN {X 0,Y 491.042,Z 1139.059,A -85,B 0,C 180,E1 15431.499,E2 15431.499} C_VEL
LIN {X 0,Y 484.646,Z 1159.746,A -85,B 0,C 180,E1 15428.989,E2 15428.989} C_VEL
LIN {X 0,Y 479.876,Z 1175.12,A -85,B 0,C 180,E1 15426.858,E2 15426.858} C_VEL
LIN {X 0,Y 475.653,Z 1188.91,A -85,B 0,C 180,E1 15424.72,E2 15424.72} C_VEL
LIN {X 0,Y 471.7,Z 1202.146,A -85,B 0,C 180,E1 15422.426,E2 15422.426} C_VEL
LIN {X 0,Y 467.471,Z 1217.266,A -85,B 0,C 180,E1 15419.464,E2 15419.464} C_VEL
LIN {X 0,Y 463.847,Z 1230.784,A -85,B 0,C 180,E1 15416.358,E2 15416.358} C_VEL
LIN {X 0,Y 461.493,Z 1240.69,A -85,B 0,C 180,E1 15413.76,E2 15413.76} C_VEL
LIN {X 0,Y 459.672,Z 1249.398,A -85,B 0,C 180,E1 15411.162,E2 15411.162} C_VEL
LIN {X 0,Y 458.211,Z 1257.328,A -85,B 0,C 180,E1 15408.441,E2 15408.441} C_VEL
LIN {X 0,Y 457.053,Z 1265.303,A -85,B 0,C 180,E1 15405.215,E2 15405.215} C_VEL
LIN {X 0,Y 456.366,Z 1271.743,A -85,B 0,C 180,E1 15401.881,E2 15401.881} C_VEL
LIN {X 0,Y 456.053,Z 1275.954,A -85,B 0,C 180,E1 15399.079,E2 15399.079} C_VEL
LIN {X 0,Y 455.959,Z 1278.916,A -85,B 0,C 180,E1 15396.417,E2 15396.417} C_VEL
LIN {X 0,Y 455.915,Z 1280.789,A -85,B 0,C 180,E1 15393.895,E2 15393.895} C_VEL
LIN {X 0,Y 455.897,Z 1281.746,A -85,B 0,C 180,E1 15391.379,E2 15391.379} C_VEL
LIN {X 0,Y 455.875,Z 1281.813,A -85,B 0,C 180,E1 15388.991,E2 15388.991} C_VEL
LIN {X 0,Y 455.914,Z 1280.991,A -85,B 0,C 180,E1 15386.476,E2 15386.476} C_VEL
LIN {X 0,Y 455.948,Z 1279.252,A -85,B 0,C 180,E1 15383.954,E2 15383.954} C_VEL
LIN {X 0,Y 456.052,Z 1276.427,A -85,B 0,C 180,E1 15381.296,E2 15381.296} C_VEL
LIN {X 0,Y 456.29,Z 1272.565,A -85,B 0,C 180,E1 15378.622,E2 15378.622} C_VEL
LIN {X 0,Y 456.732,Z 1267.896,A -85,B 0,C 180,E1 15376.062,E2 15376.062} C_VEL
LIN {X 0,Y 457.501,Z 1261.922,A -85,B 0,C 180,E1 15373.36,E2 15373.36} C_VEL
LIN {X 0,Y 458.836,Z 1253.743,A -85,B 0,C 180,E1 15370.256,E2 15370.256} C_VEL
LIN {X 0,Y 460.997,Z 1242.954,A -85,B 0,C 180,E1 15366.875,E2 15366.875} C_VEL
LIN {X 0,Y 463.38,Z 1232.751,A -85,B 0,C 180,E1 15364.134,E2 15364.134} C_VEL
LIN {X 0,Y 466.157,Z 1221.883,A -85,B 0,C 180,E1 15361.561,E2 15361.561} C_VEL
LIN {X 0,Y 469.828,Z 1208.763,A -85,B 0,C 180,E1 15358.82,E2 15358.82} C_VEL
LIN {X 0,Y 474.731,Z 1191.953,A -85,B 0,C 180,E1 15355.778,E2 15355.778} C_VEL
LIN {X 0,Y 479.234,Z 1177.165,A -85,B 0,C 180,E1 15353.445,E2 15353.445} C_VEL
LIN {X 0,Y 483.916,Z 1162.008,A -85,B 0,C 180,E1 15351.313,E2 15351.313} C_VEL
LIN {X 0,Y 489.274,Z 1144.755,A -85,B 0,C 180,E1 15349.157,E2 15349.157} C_VEL
LIN {X 0,Y 496.063,Z 1122.382,A -85,B 0,C 180,E1 15346.737,E2 15346.737} C_VEL
LIN {X 0,Y 501.38,Z 1104.241,A -85,B 0,C 180,E1 15345.033,E2 15345.033} C_VEL
LIN {X 0,Y 506.378,Z 1086.533,A -85,B 0,C 180,E1 15343.556,E2 15343.556} C_VEL
LIN {X 0,Y 511.379,Z 1067.868,A -85,B 0,C 180,E1 15342.177,E2 15342.177} C_VEL
LIN {X 0,Y 517.109,Z 1045.146,A -85,B 0,C 180,E1 15340.712,E2 15340.712} C_VEL
LIN {X 0,Y 522.858,Z 1019.507,A -85,B 0,C 180,E1 15339.325,E2 15339.325} C_VEL
LIN {X 0,Y 526.946,Z 999.331,A -85,B 0,C 180,E1 15338.4,E2 15338.4} C_VEL
LIN {X 0,Y 530.663,Z 978.787,A -85,B 0,C 180,E1 15337.596,E2 15337.596} C_VEL
LIN {X 0,Y 534.005,Z 957.646,A -85,B 0,C 180,E1 15336.902,E2 15336.902} C_VEL
LIN {X 0,Y 537.163,Z 933.916,A -85,B 0,C 180,E1 15336.269,E2 15336.269} C_VEL
LIN {X 0,Y 540.031,Z 904.65,A -85,B 0,C 180,E1 15335.688,E2 15335.688} C_VEL
LIN {X 0,Y 543.53,Z 838.394,A -85,B 0,C 180,E1 15334.663,E2 15334.663} C_VEL
LIN {X 0,Y 554.635,Z 621.494,A -85,B 0,C 180,E1 15331.351,E2 15331.351} C_VEL
LIN {X 0,Y 558.094,Z 556.51,A -85,B 0,C 180,E1 15330.347,E2 15330.347} C_VEL
LIN {X 0,Y 548.137,Z 540.877,A -85,B 0,C 180,E1 15328.105,E2 15328.105} C_VEL
LIN {X 0,Y 539.418,Z 527.859,A -85,B 0,C 180,E1 15325.942,E2 15325.942} C_VEL
LIN {X 0,Y 529.761,Z 514.212,A -85,B 0,C 180,E1 15323.263,E2 15323.263} C_VEL
LIN {X 0,Y 526.287,Z 509.77,A -85,B 0,C 180,E1 15322.215,E2 15322.215} C_VEL
LIN {X 0,Y 522.247,Z 504.73,A -85,B 0,C 180,E1 15320.921,E2 15320.921} C_VEL
LIN {X 0,Y 517.708,Z 499.113,A -85,B 0,C 180,E1 15319.344,E2 15319.344} C_VEL
LIN {X 0,Y 513.927,Z 494.369,A -85,B 0,C 180,E1 15317.903,E2 15317.903} C_VEL
LIN {X 0,Y 509.756,Z 489.745,A -85,B 0,C 180,E1 15316.173,E2 15316.173} C_VEL
LIN {X 0,Y 508.345,Z 487.735,A -85,B 0,C 180,E1 15315.516,E2 15315.516} C_VEL
LIN {X 0,Y 504.828,Z 484.1,A -85,B 0,C 180,E1 15313.808,E2 15313.808} C_VEL
LIN {X 0,Y 503.365,Z 481.702,A -85,B 0,C 180,E1 15312.971,E2 15312.971} C_VEL
LIN {X 0,Y 500.113,Z 479.064,A -85,B 0,C 180,E1 15311.066,E2 15311.066} C_VEL
LIN {X 0,Y 498.044,Z 475.338,A -85,B 0,C 180,E1 15309.476,E2 15309.476} C_VEL
LIN {X 0,Y 494.176,Z 472.541,A -85,B 0,C 180,E1 15305.923,E2 15305.923} C_VEL
LIN {X 0,Y 492.643,Z 468.777,A -85,B 0,C 180,E1 15303.025,E2 15303.025} C_VEL
LIN {X 0,Y 492.762,Z 468.873,A -85,B 0,C 180,E1 15296.51,E2 15296.51} C_VEL
LIN {X 0,Y 494.209,Z 472.521,A -85,B 0,C 180,E1 15293.844,E2 15293.844} C_VEL
LIN {X 0,Y 497.931,Z 475.306,A -85,B 0,C 180,E1 15290.406,E2 15290.406} C_VEL
LIN {X 0,Y 498.491,Z 476.255,A -85,B 0,C 180,E1 15289.95,E2 15289.95} C_VEL
LIN {X 0,Y 500.686,Z 479.697,A -85,B 0,C 180,E1 15288.363,E2 15288.363} C_VEL
LIN {X 0,Y 503.723,Z 482.131,A -85,B 0,C 180,E1 15286.629,E2 15286.629} C_VEL
LIN {X 0,Y 506.625,Z 486.3,A -85,B 0,C 180,E1 15285.075,E2 15285.075} C_VEL
LIN {X 0,Y 509.016,Z 488.501,A -85,B 0,C 180,E1 15283.979,E2 15283.979} C_VEL
LIN {X 0,Y 512.374,Z 492.844,A -85,B 0,C 180,E1 15282.511,E2 15282.511} C_VEL
LIN {X 0,Y 514.144,Z 494.643,A -85,B 0,C 180,E1 15281.812,E2 15281.812} C_VEL
LIN {X 0,Y 517.956,Z 499.295,A -85,B 0,C 180,E1 15280.373,E2 15280.373} C_VEL
LIN {X 0,Y 524.181,Z 507.094,A -85,B 0,C 180,E1 15278.251,E2 15278.251} C_VEL
LIN {X 0,Y 528.841,Z 512.976,A -85,B 0,C 180,E1 15276.812,E2 15276.812} C_VEL
LIN {X 0,Y 535.801,Z 521.84,A -85,B 0,C 180,E1 15274.848,E2 15274.848} C_VEL
LIN {X 0,Y 545.231,Z 534.633,A -85,B 0,C 180,E1 15272.445,E2 15272.445} C_VEL
LIN {X 0,Y 553.057,Z 545.749,A -85,B 0,C 180,E1 15270.633,E2 15270.633} C_VEL
LIN {X 0,Y 558.128,Z 553.995,A -85,B 0,C 180,E1 15269.511,E2 15269.511} C_VEL
LIN {X 0,Y 546.566,Z 774.311,A -85,B 0,C 180,E1 15266.139,E2 15266.139} C_VEL
LIN {X 0,Y 540.309,Z 895.949,A -85,B 0,C 180,E1 15264.274,E2 15264.274} C_VEL
LIN {X 0,Y 537.851,Z 923.031,A -85,B 0,C 180,E1 15263.753,E2 15263.753} C_VEL
LIN {X 0,Y 534.367,Z 949.691,A -85,B 0,C 180,E1 15263.049,E2 15263.049} C_VEL
LIN {X 0,Y 531.053,Z 970.943,A -85,B 0,C 180,E1 15262.35,E2 15262.35} C_VEL
LIN {X 0,Y 527.362,Z 991.502,A -85,B 0,C 180,E1 15261.543,E2 15261.543} C_VEL
LIN {X 0,Y 523.06,Z 1012.79,A -85,B 0,C 180,E1 15260.562,E2 15260.562} C_VEL
LIN {X 0,Y 517.1,Z 1039.077,A -85,B 0,C 180,E1 15259.119,E2 15259.119} C_VEL
LIN {X 0,Y 511.622,Z 1060.719,A -85,B 0,C 180,E1 15257.709,E2 15257.709} C_VEL
LIN {X 0,Y 506.672,Z 1079.087,A -85,B 0,C 180,E1 15256.342,E2 15256.342} C_VEL
LIN {X 0,Y 501.703,Z 1096.574,A -85,B 0,C 180,E1 15254.873,E2 15254.873} C_VEL
LIN {X 0,Y 496.161,Z 1115.338,A -85,B 0,C 180,E1 15253.094,E2 15253.094} C_VEL
LIN {X 0,Y 489.355,Z 1137.365,A -85,B 0,C 180,E1 15250.68,E2 15250.68} C_VEL
LIN {X 0,Y 484.148,Z 1153.924,A -85,B 0,C 180,E1 15248.59,E2 15248.59} C_VEL
LIN {X 0,Y 479.461,Z 1168.86,A -85,B 0,C 180,E1 15246.469,E2 15246.469} C_VEL
LIN {X 0,Y 474.466,Z 1185.095,A -85,B 0,C 180,E1 15243.868,E2 15243.868} C_VEL
LIN {X 0,Y 472.731,Z 1190.74,A -85,B 0,C 180,E1 15242.858,E2 15242.858} C_VEL
LIN {X 0,Y 470.529,Z 1195.134,A -85,B 0,C 180,E1 15242.124,E2 15242.124} C_VEL
LIN {X 0,Y 461.553,Z 1206.745,A -85,B 0,C 180,E1 15240.239,E2 15240.239} C_VEL
LIN {X 0,Y 459.857,Z 1210.074,A -85,B 0,C 180,E1 15239.554,E2 15239.554} C_VEL
LIN {X 0,Y 456.33,Z 1222.373,A -85,B 0,C 180,E1 15236.62,E2 15236.62} C_VEL
LIN {X 0,Y 453.902,Z 1231.823,A -85,B 0,C 180,E1 15234.053,E2 15234.053} C_VEL
LIN {X 0,Y 451.867,Z 1240.754,A -85,B 0,C 180,E1 15231.281,E2 15231.281} C_VEL
LIN {X 0,Y 450.041,Z 1250.21,A -85,B 0,C 180,E1 15227.858,E2 15227.858} C_VEL
LIN {X 0,Y 448.907,Z 1257.444,A -85,B 0,C 180,E1 15224.581,E2 15224.581} C_VEL
LIN {X 0,Y 448.362,Z 1262.591,A -85,B 0,C 180,E1 15221.712,E2 15221.712} C_VEL
LIN {X 0,Y 448.062,Z 1266.439,A -85,B 0,C 180,E1 15218.99,E2 15218.99} C_VEL
LIN {X 0,Y 447.959,Z 1269.267,A -85,B 0,C 180,E1 15216.283,E2 15216.283} C_VEL
LIN {X 0,Y 447.917,Z 1271.03,A -85,B 0,C 180,E1 15213.715,E2 15213.715} C_VEL
LIN {X 0,Y 447.889,Z 1271.896,A -85,B 0,C 180,E1 15211.155,E2 15211.155} C_VEL
LIN {X 0,Y 447.895,Z 1271.868,A -85,B 0,C 180,E1 15208.597,E2 15208.597} C_VEL
LIN {X 0,Y 447.917,Z 1270.947,A -85,B 0,C 180,E1 15206.036,E2 15206.036} C_VEL
LIN {X 0,Y 447.965,Z 1269.028,A -85,B 0,C 180,E1 15203.353,E2 15203.353} C_VEL
LIN {X 0,Y 448.066,Z 1266.085,A -85,B 0,C 180,E1 15200.629,E2 15200.629} C_VEL
LIN {X 0,Y 448.451,Z 1261.721,A -85,B 0,C 180,E1 15197.645,E2 15197.645} C_VEL
LIN {X 0,Y 449.335,Z 1254.642,A -85,B 0,C 180,E1 15193.987,E2 15193.987} C_VEL
LIN {X 0,Y 450.548,Z 1247.323,A -85,B 0,C 180,E1 15190.965,E2 15190.965} C_VEL
LIN {X 0,Y 452.156,Z 1239.437,A -85,B 0,C 180,E1 15188.196,E2 15188.196} C_VEL
LIN {X 0,Y 454.407,Z 1229.865,A -85,B 0,C 180,E1 15185.292,E2 15185.292} C_VEL
LIN {X 0,Y 458.107,Z 1216.057,A -85,B 0,C 180,E1 15181.735,E2 15181.735} C_VEL
LIN {X 0,Y 461.593,Z 1204.037,A -85,B 0,C 180,E1 15179.071,E2 15179.071} C_VEL
LIN {X 0,Y 465.454,Z 1191.649,A -85,B 0,C 180,E1 15176.643,E2 15176.643} C_VEL
LIN {X 0,Y 470.117,Z 1177.196,A -85,B 0,C 180,E1 15174.13,E2 15174.13} C_VEL
LIN {X 0,Y 476.408,Z 1157.848,A -85,B 0,C 180,E1 15171.215,E2 15171.215} C_VEL
LIN {X 0,Y 481.751,Z 1141.445,A -85,B 0,C 180,E1 15169.069,E2 15169.069} C_VEL
LIN {X 0,Y 486.97,Z 1125.281,A -85,B 0,C 180,E1 15167.192,E2 15167.192} C_VEL
LIN {X 0,Y 492.702,Z 1107.127,A -85,B 0,C 180,E1 15165.324,E2 15165.324} C_VEL
LIN {X 0,Y 499.903,Z 1083.179,A -85,B 0,C 180,E1 15163.2,E2 15163.2} C_VEL
LIN {X 0,Y 505.442,Z 1063.451,A -85,B 0,C 180,E1 15161.695,E2 15161.695} C_VEL
LIN {X 0,Y 510.467,Z 1044.365,A -85,B 0,C 180,E1 15160.418,E2 15160.418} C_VEL
LIN {X 0,Y 515.482,Z 1023.871,A -85,B 0,C 180,E1 15159.224,E2 15159.224} C_VEL
LIN {X 0,Y 520.881,Z 999.569,A -85,B 0,C 180,E1 15158.01,E2 15158.01} C_VEL
LIN {X 0,Y 525.633,Z 974.31,A -85,B 0,C 180,E1 15156.979,E2 15156.979} C_VEL
LIN {X 0,Y 529.129,Z 952.935,A -85,B 0,C 180,E1 15156.256,E2 15156.256} C_VEL
LIN {X 0,Y 532.1,Z 931.51,A -85,B 0,C 180,E1 15155.663,E2 15155.663} C_VEL
LIN {X 0,Y 534.667,Z 908.51,A -85,B 0,C 180,E1 15155.158,E2 15155.158} C_VEL
LIN {X 0,Y 537.123,Z 872.623,A -85,B 0,C 180,E1 15154.562,E2 15154.562} C_VEL
LIN {X 0,Y 548.777,Z 651.348,A -85,B 0,C 180,E1 15151.177,E2 15151.177} C_VEL
LIN {X 0,Y 553.892,Z 558.206,A -85,B 0,C 180,E1 15149.735,E2 15149.735} C_VEL
LIN {X 0,Y 546.541,Z 546.947,A -85,B 0,C 180,E1 15148.046,E2 15148.046} C_VEL
LIN {X 0,Y 536.678,Z 533.187,A -85,B 0,C 180,E1 15145.58,E2 15145.58} C_VEL
LIN {X 0,Y 528.229,Z 522.109,A -85,B 0,C 180,E1 15143.216,E2 15143.216} C_VEL
LIN {X 0,Y 523.963,Z 516.684,A -85,B 0,C 180,E1 15141.906,E2 15141.906} C_VEL
LIN {X 0,Y 520.166,Z 511.902,A -85,B 0,C 180,E1 15140.655,E2 15140.655} C_VEL
LIN {X 0,Y 515.869,Z 506.509,A -85,B 0,C 180,E1 15139.121,E2 15139.121} C_VEL
LIN {X 0,Y 511.498,Z 501.116,A -85,B 0,C 180,E1 15137.403,E2 15137.403} C_VEL
LIN {X 0,Y 507.989,Z 496.966,A -85,B 0,C 180,E1 15135.879,E2 15135.879} C_VEL
LIN {X 0,Y 506.834,Z 495.404,A -85,B 0,C 180,E1 15135.329,E2 15135.329} C_VEL
LIN {X 0,Y 503.314,Z 491.569,A -85,B 0,C 180,E1 15133.558,E2 15133.558} C_VEL
LIN {X 0,Y 501.977,Z 489.467,A -85,B 0,C 180,E1 15132.774,E2 15132.774} C_VEL
LIN {X 0,Y 498.753,Z 486.681,A -85,B 0,C 180,E1 15130.804,E2 15130.804} C_VEL
LIN {X 0,Y 496.834,Z 483.204,A -85,B 0,C 180,E1 15129.265,E2 15129.265} C_VEL
LIN {X 0,Y 492.992,Z 480.242,A -85,B 0,C 180,E1 15125.47,E2 15125.47} C_VEL
LIN {X 0,Y 491.693,Z 476.736,A -85,B 0,C 180,E1 15122.564,E2 15122.564} C_VEL
LIN {X 0,Y 491.771,Z 476.822,A -85,B 0,C 180,E1 15117.32,E2 15117.32} C_VEL
LIN {X 0,Y 493.695,Z 481.13,A -85,B 0,C 180,E1 15113.721,E2 15113.721} C_VEL
LIN {X 0,Y 497.103,Z 483.566,A -85,B 0,C 180,E1 15110.623,E2 15110.623} C_VEL
LIN {X 0,Y 499.316,Z 487.409,A -85,B 0,C 180,E1 15108.916,E2 15108.916} C_VEL
LIN {X 0,Y 502.447,Z 490.062,A -85,B 0,C 180,E1 15107.063,E2 15107.063} C_VEL
LIN {X 0,Y 505.639,Z 494.423,A -85,B 0,C 180,E1 15105.338,E2 15105.338} C_VEL
LIN {X 0,Y 507.517,Z 496.225,A -85,B 0,C 180,E1 15104.458,E2 15104.458} C_VEL
LIN {X 0,Y 510.939,Z 500.647,A -85,B 0,C 180,E1 15102.93,E2 15102.93} C_VEL
LIN {X 0,Y 512.539,Z 502.349,A -85,B 0,C 180,E1 15102.282,E2 15102.282} C_VEL
LIN {X 0,Y 516.439,Z 507.047,A -85,B 0,C 180,E1 15100.783,E2 15100.783} C_VEL
LIN {X 0,Y 522.566,Z 514.962,A -85,B 0,C 180,E1 15098.652,E2 15098.652} C_VEL
LIN {X 0,Y 526.836,Z 520.372,A -85,B 0,C 180,E1 15097.309,E2 15097.309} C_VEL
LIN {X 0,Y 534.975,Z 531.855,A -85,B 0,C 180,E1 15094.954,E2 15094.954} C_VEL
LIN {X 0,Y 543.801,Z 545.086,A -85,B 0,C 180,E1 15092.663,E2 15092.663} C_VEL
LIN {X 0,Y 553.899,Z 560.989,A -85,B 0,C 180,E1 15090.302,E2 15090.302} C_VEL
LIN {X 0,Y 542.697,Z 767.938,A -85,B 0,C 180,E1 15087.118,E2 15087.118} C_VEL
LIN {X 0,Y 535.566,Z 902.547,A -85,B 0,C 180,E1 15085.047,E2 15085.047} C_VEL
LIN {X 0,Y 533.048,Z 929.459,A -85,B 0,C 180,E1 15084.535,E2 15084.535} C_VEL
LIN {X 0,Y 529.448,Z 956.193,A -85,B 0,C 180,E1 15083.841,E2 15083.841} C_VEL
LIN {X 0,Y 525.995,Z 977.53,A -85,B 0,C 180,E1 15083.15,E2 15083.15} C_VEL
LIN {X 0,Y 522.207,Z 998.048,A -85,B 0,C 180,E1 15082.352,E2 15082.352} C_VEL
LIN {X 0,Y 517.945,Z 1018.51,A -85,B 0,C 180,E1 15081.422,E2 15081.422} C_VEL
LIN {X 0,Y 512.494,Z 1042.426,A -85,B 0,C 180,E1 15080.142,E2 15080.142} C_VEL
LIN {X 0,Y 506.319,Z 1066.308,A -85,B 0,C 180,E1 15078.62,E2 15078.62} C_VEL
LIN {X 0,Y 501.114,Z 1085.111,A -85,B 0,C 180,E1 15077.239,E2 15077.239} C_VEL
LIN {X 0,Y 495.927,Z 1102.867,A -85,B 0,C 180,E1 15075.764,E2 15075.764} C_VEL
LIN {X 0,Y 490.545,Z 1120.562,A -85,B 0,C 180,E1 15074.107,E2 15074.107} C_VEL
LIN {X 0,Y 484.151,Z 1141.144,A -85,B 0,C 180,E1 15071.914,E2 15071.914} C_VEL
LIN {X 0,Y 477.84,Z 1160.586,A -85,B 0,C 180,E1 15069.497,E2 15069.497} C_VEL
LIN {X 0,Y 472.898,Z 1175.873,A -85,B 0,C 180,E1 15067.343,E2 15067.343} C_VEL
LIN {X 0,Y 468.514,Z 1189.608,A -85,B 0,C 180,E1 15065.175,E2 15065.175} C_VEL
LIN {X 0,Y 464.191,Z 1203.464,A -85,B 0,C 180,E1 15062.723,E2 15062.723} C_VEL
LIN {X 0,Y 459.286,Z 1220.087,A -85,B 0,C 180,E1 15059.324,E2 15059.324} C_VEL
LIN {X 0,Y 456.207,Z 1231.211,A -85,B 0,C 180,E1 15056.694,E2 15056.694} C_VEL
LIN {X 0,Y 453.751,Z 1241.061,A -85,B 0,C 180,E1 15054.053,E2 15054.053} C_VEL
LIN {X 0,Y 451.844,Z 1249.715,A -85,B 0,C 180,E1 15051.411,E2 15051.411} C_VEL
LIN {X 0,Y 450.193,Z 1258.306,A -85,B 0,C 180,E1 15048.379,E2 15048.379} C_VEL
LIN {X 0,Y 448.934,Z 1266.537,A -85,B 0,C 180,E1 15044.836,E2 15044.836} C_VEL
LIN {X 0,Y 448.381,Z 1271.863,A -85,B 0,C 180,E1 15041.965,E2 15041.965} C_VEL
LIN {X 0,Y 448.056,Z 1275.865,A -85,B 0,C 180,E1 15039.242,E2 15039.242} C_VEL
LIN {X 0,Y 447.961,Z 1278.828,A -85,B 0,C 180,E1 15036.532,E2 15036.532} C_VEL
LIN {X 0,Y 447.916,Z 1280.701,A -85,B 0,C 180,E1 15033.964,E2 15033.964} C_VEL
LIN {X 0,Y 447.899,Z 1281.658,A -85,B 0,C 180,E1 15031.403,E2 15031.403} C_VEL
LIN {X 0,Y 447.877,Z 1281.725,A -85,B 0,C 180,E1 15028.973,E2 15028.973} C_VEL
LIN {X 0,Y 447.915,Z 1280.903,A -85,B 0,C 180,E1 15026.413,E2 15026.413} C_VEL
LIN {X 0,Y 447.951,Z 1279.164,A -85,B 0,C 180,E1 15023.846,E2 15023.846} C_VEL
LIN {X 0,Y 448.054,Z 1276.339,A -85,B 0,C 180,E1 15021.139,E2 15021.139} C_VEL
LIN {X 0,Y 448.301,Z 1272.685,A -85,B 0,C 180,E1 15018.547,E2 15018.547} C_VEL
LIN {X 0,Y 448.758,Z 1268.063,A -85,B 0,C 180,E1 15015.941,E2 15015.941} C_VEL
LIN {X 0,Y 449.521,Z 1262.443,A -85,B 0,C 180,E1 15013.322,E2 15013.322} C_VEL
LIN {X 0,Y 450.705,Z 1255.379,A -85,B 0,C 180,E1 15010.539,E2 15010.539} C_VEL
LIN {X 0,Y 452.744,Z 1245.609,A -85,B 0,C 180,E1 15007.261,E2 15007.261} C_VEL
LIN {X 0,Y 455.571,Z 1233.781,A -85,B 0,C 180,E1 15003.96,E2 15003.96} C_VEL
LIN {X 0,Y 458.46,Z 1222.946,A -85,B 0,C 180,E1 15001.324,E2 15001.324} C_VEL
LIN {X 0,Y 461.894,Z 1211.072,A -85,B 0,C 180,E1 14998.769,E2 14998.769} C_VEL
LIN {X 0,Y 466.411,Z 1196.373,A -85,B 0,C 180,E1 14995.974,E2 14995.974} C_VEL
LIN {X 0,Y 471.844,Z 1179.152,A -85,B 0,C 180,E1 14993.149,E2 14993.149} C_VEL
LIN {X 0,Y 476.785,Z 1163.774,A -85,B 0,C 180,E1 14990.933,E2 14990.933} C_VEL
LIN {X 0,Y 481.787,Z 1148.224,A -85,B 0,C 180,E1 14988.937,E2 14988.937} C_VEL
LIN {X 0,Y 487.274,Z 1131.02,A -85,B 0,C 180,E1 14986.975,E2 14986.975} C_VEL
LIN {X 0,Y 494.221,Z 1108.645,A -85,B 0,C 180,E1 14984.753,E2 14984.753} C_VEL
LIN {X 0,Y 500.079,Z 1088.65,A -85,B 0,C 180,E1 14983.044,E2 14983.044} C_VEL
LIN {X 0,Y 505.227,Z 1070.161,A -85,B 0,C 180,E1 14981.652,E2 14981.652} C_VEL
LIN {X 0,Y 510.141,Z 1051.369,A -85,B 0,C 180,E1 14980.404,E2 14980.404} C_VEL
LIN {X 0,Y 515.07,Z 1031.146,A -85,B 0,C 180,E1 14979.233,E2 14979.233} C_VEL
LIN {X 0,Y 520.703,Z 1005.671,A -85,B 0,C 180,E1 14977.974,E2 14977.974} C_VEL
LIN {X 0,Y 525.248,Z 981.651,A -85,B 0,C 180,E1 14977.003,E2 14977.003} C_VEL
LIN {X 0,Y 528.812,Z 960.031,A -85,B 0,C 180,E1 14976.277,E2 14976.277} C_VEL
LIN {X 0,Y 531.794,Z 938.775,A -85,B 0,C 180,E1 14975.693,E2 14975.693} C_VEL
LIN {X 0,Y 534.36,Z 916.192,A -85,B 0,C 180,E1 14975.201,E2 14975.201} C_VEL
LIN {X 0,Y 536.715,Z 883.159,A -85,B 0,C 180,E1 14974.644,E2 14974.644} C_VEL
LIN {X 0,Y 548.325,Z 661.262,A -85,B 0,C 180,E1 14971.251,E2 14971.251} C_VEL
LIN {X 0,Y 553.765,Z 560.841,A -85,B 0,C 180,E1 14969.687,E2 14969.687} C_VEL
LIN {X 0,Y 542.36,Z 542.791,A -85,B 0,C 180,E1 14967,E2 14967} C_VEL
LIN {X 0,Y 533.416,Z 529.77,A -85,B 0,C 180,E1 14964.65,E2 14964.65} C_VEL
LIN {X 0,Y 525.327,Z 518.21,A -85,B 0,C 180,E1 14962.258,E2 14962.258} C_VEL
LIN {X 0,Y 519.981,Z 511.741,A -85,B 0,C 180,E1 14960.532,E2 14960.532} C_VEL
LIN {X 0,Y 515.858,Z 506.521,A -85,B 0,C 180,E1 14959.063,E2 14959.063} C_VEL
LIN {X 0,Y 511.465,Z 501.104,A -85,B 0,C 180,E1 14957.345,E2 14957.345} C_VEL
LIN {X 0,Y 507.938,Z 496.925,A -85,B 0,C 180,E1 14955.822,E2 14955.822} C_VEL
LIN {X 0,Y 506.897,Z 495.446,A -85,B 0,C 180,E1 14955.327,E2 14955.327} C_VEL
LIN {X 0,Y 503.332,Z 491.644,A -85,B 0,C 180,E1 14953.557,E2 14953.557} C_VEL
LIN {X 0,Y 501.986,Z 489.476,A -85,B 0,C 180,E1 14952.774,E2 14952.774} C_VEL
LIN {X 0,Y 498.721,Z 486.646,A -85,B 0,C 180,E1 14950.805,E2 14950.805} C_VEL
LIN {X 0,Y 496.765,Z 483.173,A -85,B 0,C 180,E1 14949.266,E2 14949.266} C_VEL
LIN {X 0,Y 493.023,Z 480.294,A -85,B 0,C 180,E1 14945.703,E2 14945.703} C_VEL
LIN {X 0,Y 491.617,Z 476.71,A -85,B 0,C 180,E1 14942.915,E2 14942.915} C_VEL
LIN {X 0,Y 491.735,Z 476.771,A -85,B 0,C 180,E1 14936.619,E2 14936.619} C_VEL
LIN {X 0,Y 493.143,Z 480.399,A -85,B 0,C 180,E1 14933.948,E2 14933.948} C_VEL
LIN {X 0,Y 497.059,Z 483.562,A -85,B 0,C 180,E1 14930.298,E2 14930.298} C_VEL
LIN {X 0,Y 499.19,Z 487.212,A -85,B 0,C 180,E1 14928.679,E2 14928.679} C_VEL
LIN {X 0,Y 502.435,Z 490.047,A -85,B 0,C 180,E1 14926.77,E2 14926.77} C_VEL
LIN {X 0,Y 505.431,Z 494.216,A -85,B 0,C 180,E1 14925.156,E2 14925.156} C_VEL
LIN {X 0,Y 507.442,Z 496.061,A -85,B 0,C 180,E1 14924.221,E2 14924.221} C_VEL
LIN {X 0,Y 510.879,Z 500.533,A -85,B 0,C 180,E1 14922.693,E2 14922.693} C_VEL
LIN {X 0,Y 512.553,Z 502.32,A -85,B 0,C 180,E1 14922.018,E2 14922.018} C_VEL
LIN {X 0,Y 516.551,Z 507.12,A -85,B 0,C 180,E1 14920.494,E2 14920.494} C_VEL
LIN {X 0,Y 521.076,Z 512.791,A -85,B 0,C 180,E1 14918.912,E2 14918.912} C_VEL
LIN {X 0,Y 529.606,Z 523.791,A -85,B 0,C 180,E1 14916.258,E2 14916.258} C_VEL
LIN {X 0,Y 539.334,Z 536.897,A -85,B 0,C 180,E1 14913.61,E2 14913.61} C_VEL
LIN {X 0,Y 548.928,Z 550.403,A -85,B 0,C 180,E1 14911.286,E2 14911.286} C_VEL
LIN {X 0,Y 553.857,Z 558.43,A -85,B 0,C 180,E1 14910.159,E2 14910.159} C_VEL
LIN {X 0,Y 541.861,Z 779.657,A -85,B 0,C 180,E1 14906.763,E2 14906.763} C_VEL
LIN {X 0,Y 535.658,Z 896.168,A -85,B 0,C 180,E1 14904.968,E2 14904.968} C_VEL
LIN {X 0,Y 533.097,Z 923.525,A -85,B 0,C 180,E1 14904.44,E2 14904.44} C_VEL
LIN {X 0,Y 529.539,Z 949.954,A -85,B 0,C 180,E1 14903.741,E2 14903.741} C_VEL
LIN {X 0,Y 526.156,Z 971.042,A -85,B 0,C 180,E1 14903.046,E2 14903.046} C_VEL
LIN {X 0,Y 522.612,Z 990.318,A -85,B 0,C 180,E1 14902.293,E2 14902.293} C_VEL
LIN {X 0,Y 518.255,Z 1011.358,A -85,B 0,C 180,E1 14901.332,E2 14901.332} C_VEL
LIN {X 0,Y 512.976,Z 1034.517,A -85,B 0,C 180,E1 14900.088,E2 14900.088} C_VEL
LIN {X 0,Y 506.591,Z 1059.198,A -85,B 0,C 180,E1 14898.509,E2 14898.509} C_VEL
LIN {X 0,Y 501.407,Z 1077.852,A -85,B 0,C 180,E1 14897.128,E2 14897.128} C_VEL
LIN {X 0,Y 496.271,Z 1095.339,A -85,B 0,C 180,E1 14895.666,E2 14895.666} C_VEL
LIN {X 0,Y 490.956,Z 1112.67,A -85,B 0,C 180,E1 14894.034,E2 14894.034} C_VEL
LIN {X 0,Y 484.785,Z 1132.301,A -85,B 0,C 180,E1 14891.935,E2 14891.935} C_VEL
LIN {X 0,Y 478.267,Z 1152.177,A -85,B 0,C 180,E1 14889.464,E2 14889.464} C_VEL
LIN {X 0,Y 473.311,Z 1167.274,A -85,B 0,C 180,E1 14887.325,E2 14887.325} C_VEL
LIN {X 0,Y 468.871,Z 1180.921,A -85,B 0,C 180,E1 14885.157,E2 14885.157} C_VEL
LIN {X 0,Y 464.444,Z 1194.848,A -85,B 0,C 180,E1 14882.672,E2 14882.672} C_VEL
LIN {X 0,Y 459.857,Z 1210.074,A -85,B 0,C 180,E1 14879.554,E2 14879.554} C_VEL
LIN {X 0,Y 457.798,Z 1213.921,A -85,B 0,C 180,E1 14878.745,E2 14878.745} C_VEL
LIN {X 0,Y 449.169,Z 1224.026,A -85,B 0,C 180,E1 14876.651,E2 14876.651} C_VEL
LIN {X 0,Y 447.674,Z 1226.967,A -85,B 0,C 180,E1 14875.917,E2 14875.917} C_VEL
LIN {X 0,Y 444.697,Z 1238.476,A -85,B 0,C 180,E1 14872.463,E2 14872.463} C_VEL
LIN {X 0,Y 442.913,Z 1246.459,A -85,B 0,C 180,E1 14869.659,E2 14869.659} C_VEL
LIN {X 0,Y 441.658,Z 1253.31,A -85,B 0,C 180,E1 14866.848,E2 14866.848} C_VEL
LIN {X 0,Y 440.83,Z 1258.794,A -85,B 0,C 180,E1 14864.183,E2 14864.183} C_VEL
LIN {X 0,Y 440.323,Z 1263.499,A -85,B 0,C 180,E1 14861.398,E2 14861.398} C_VEL
LIN {X 0,Y 440.031,Z 1267.476,A -85,B 0,C 180,E1 14858.365,E2 14858.365} C_VEL
LIN {X 0,Y 439.928,Z 1270.513,A -85,B 0,C 180,E1 14854.958,E2 14854.958} C_VEL
LIN {X 0,Y 439.908,Z 1271.871,A -85,B 0,C 180,E1 14851.827,E2 14851.827} C_VEL
LIN {X 0,Y 439.87,Z 1272.046,A -85,B 0,C 180,E1 14849.092,E2 14849.092} C_VEL
LIN {X 0,Y 439.916,Z 1271.236,A -85,B 0,C 180,E1 14846.355,E2 14846.355} C_VEL
LIN {X 0,Y 439.963,Z 1269.441,A -85,B 0,C 180,E1 14843.61,E2 14843.61} C_VEL
LIN {X 0,Y 440.066,Z 1266.646,A -85,B 0,C 180,E1 14840.853,E2 14840.853} C_VEL
LIN {X 0,Y 440.378,Z 1262.902,A -85,B 0,C 180,E1 14838.126,E2 14838.126} C_VEL
LIN {X 0,Y 440.895,Z 1258.222,A -85,B 0,C 180,E1 14835.425,E2 14835.425} C_VEL
LIN {X 0,Y 441.832,Z 1252.328,A -85,B 0,C 180,E1 14832.624,E2 14832.624} C_VEL
LIN {X 0,Y 443.567,Z 1243.543,A -85,B 0,C 180,E1 14829.14,E2 14829.14} C_VEL
LIN {X 0,Y 445.992,Z 1233.14,A -85,B 0,C 180,E1 14825.783,E2 14825.783} C_VEL
LIN {X 0,Y 448.59,Z 1223.462,A -85,B 0,C 180,E1 14823.074,E2 14823.074} C_VEL
LIN {X 0,Y 451.764,Z 1212.73,A -85,B 0,C 180,E1 14820.431,E2 14820.431} C_VEL
LIN {X 0,Y 456.248,Z 1198.645,A -85,B 0,C 180,E1 14817.382,E2 14817.382} C_VEL
LIN {X 0,Y 461.369,Z 1183.056,A -85,B 0,C 180,E1 14814.498,E2 14814.498} C_VEL
LIN {X 0,Y 466.215,Z 1168.761,A -85,B 0,C 180,E1 14812.172,E2 14812.172} C_VEL
LIN {X 0,Y 471.334,Z 1153.79,A -85,B 0,C 180,E1 14810.007,E2 14810.007} C_VEL
LIN {X 0,Y 477.151,Z 1136.741,A -85,B 0,C 180,E1 14807.823,E2 14807.823} C_VEL
LIN {X 0,Y 484.341,Z 1115.014,A -85,B 0,C 180,E1 14805.417,E2 14805.417} C_VEL
LIN {X 0,Y 490.09,Z 1096.944,A -85,B 0,C 180,E1 14803.684,E2 14803.684} C_VEL
LIN {X 0,Y 495.38,Z 1079.602,A -85,B 0,C 180,E1 14802.212,E2 14802.212} C_VEL
LIN {X 0,Y 500.479,Z 1061.916,A -85,B 0,C 180,E1 14800.879,E2 14800.879} C_VEL
LIN {X 0,Y 505.807,Z 1042.161,A -85,B 0,C 180,E1 14799.568,E2 14799.568} C_VEL
LIN {X 0,Y 511.891,Z 1017.73,A -85,B 0,C 180,E1 14798.176,E2 14798.176} C_VEL
LIN {X 0,Y 517.17,Z 993.242,A -85,B 0,C 180,E1 14797.023,E2 14797.023} C_VEL
LIN {X 0,Y 521.141,Z 972.516,A -85,B 0,C 180,E1 14796.2,E2 14796.2} C_VEL
LIN {X 0,Y 524.641,Z 951.473,A -85,B 0,C 180,E1 14795.499,E2 14795.499} C_VEL
LIN {X 0,Y 527.813,Z 928.851,A -85,B 0,C 180,E1 14794.885,E2 14794.885} C_VEL
LIN {X 0,Y 530.915,Z 899.513,A -85,B 0,C 180,E1 14794.283,E2 14794.283} C_VEL
LIN {X 0,Y 533.994,Z 846.412,A -85,B 0,C 180,E1 14793.448,E2 14793.448} C_VEL
LIN {X 0,Y 546.016,Z 627.339,A -85,B 0,C 180,E1 14790.082,E2 14790.082} C_VEL
LIN {X 0,Y 549.626,Z 562.581,A -85,B 0,C 180,E1 14789.061,E2 14789.061} C_VEL
LIN {X 0,Y 543.423,Z 553.136,A -85,B 0,C 180,E1 14787.595,E2 14787.595} C_VEL
LIN {X 0,Y 534.292,Z 540.216,A -85,B 0,C 180,E1 14785.258,E2 14785.258} C_VEL
LIN {X 0,Y 526.053,Z 529.262,A -85,B 0,C 180,E1 14782.903,E2 14782.903} C_VEL
LIN {X 0,Y 521.852,Z 523.854,A -85,B 0,C 180,E1 14781.585,E2 14781.585} C_VEL
LIN {X 0,Y 518.269,Z 519.277,A -85,B 0,C 180,E1 14780.38,E2 14780.38} C_VEL
LIN {X 0,Y 514.036,Z 513.912,A -85,B 0,C 180,E1 14778.838,E2 14778.838} C_VEL
LIN {X 0,Y 509.869,Z 508.69,A -85,B 0,C 180,E1 14777.166,E2 14777.166} C_VEL
LIN {X 0,Y 506.309,Z 504.33,A -85,B 0,C 180,E1 14775.58,E2 14775.58} C_VEL
LIN {X 0,Y 505.16,Z 502.927,A -85,B 0,C 180,E1 14775.028,E2 14775.028} C_VEL
LIN {X 0,Y 501.643,Z 498.804,A -85,B 0,C 180,E1 14773.193,E2 14773.193} C_VEL
LIN {X 0,Y 500.61,Z 497.236,A -85,B 0,C 180,E1 14772.575,E2 14772.575} C_VEL
LIN {X 0,Y 497.378,Z 494.26,A -85,B 0,C 180,E1 14770.541,E2 14770.541} C_VEL
LIN {X 0,Y 495.717,Z 491.098,A -85,B 0,C 180,E1 14769.169,E2 14769.169} C_VEL
LIN {X 0,Y 491.935,Z 488.121,A -85,B 0,C 180,E1 14765.365,E2 14765.365} C_VEL
LIN {X 0,Y 490.677,Z 484.672,A -85,B 0,C 180,E1 14762.453,E2 14762.453} C_VEL
LIN {X 0,Y 490.78,Z 484.901,A -85,B 0,C 180,E1 14757.314,E2 14757.314} C_VEL
LIN {X 0,Y 492.722,Z 489.106,A -85,B 0,C 180,E1 14753.709,E2 14753.709} C_VEL
LIN {X 0,Y 495.907,Z 491.421,A -85,B 0,C 180,E1 14750.776,E2 14750.776} C_VEL
LIN {X 0,Y 498.173,Z 495.304,A -85,B 0,C 180,E1 14749.008,E2 14749.008} C_VEL
LIN {X 0,Y 501.077,Z 497.782,A -85,B 0,C 180,E1 14747.261,E2 14747.261} C_VEL
LIN {X 0,Y 504.332,Z 502.225,A -85,B 0,C 180,E1 14745.475,E2 14745.475} C_VEL
LIN {X 0,Y 506.065,Z 503.97,A -85,B 0,C 180,E1 14744.647,E2 14744.647} C_VEL
LIN {X 0,Y 509.582,Z 508.458,A -85,B 0,C 180,E1 14743.059,E2 14743.059} C_VEL
LIN {X 0,Y 511.151,Z 510.311,A -85,B 0,C 180,E1 14742.409,E2 14742.409} C_VEL
LIN {X 0,Y 515.656,Z 515.949,A -85,B 0,C 180,E1 14740.665,E2 14740.665} C_VEL
LIN {X 0,Y 520.635,Z 522.324,A -85,B 0,C 180,E1 14738.923,E2 14738.923} C_VEL
LIN {X 0,Y 524.929,Z 527.854,A -85,B 0,C 180,E1 14737.548,E2 14737.548} C_VEL
LIN {X 0,Y 532.791,Z 539.154,A -85,B 0,C 180,E1 14735.23,E2 14735.23} C_VEL
LIN {X 0,Y 541.219,Z 551.97,A -85,B 0,C 180,E1 14732.998,E2 14732.998} C_VEL
LIN {X 0,Y 549.702,Z 565.615,A -85,B 0,C 180,E1 14730.954,E2 14730.954} C_VEL
LIN {X 0,Y 537.662,Z 781.005,A -85,B 0,C 180,E1 14727.635,E2 14727.635} C_VEL
LIN {X 0,Y 530.988,Z 902.692,A -85,B 0,C 180,E1 14725.754,E2 14725.754} C_VEL
LIN {X 0,Y 528.336,Z 930.148,A -85,B 0,C 180,E1 14725.229,E2 14725.229} C_VEL
LIN {X 0,Y 524.675,Z 956.44,A -85,B 0,C 180,E1 14724.543,E2 14724.543} C_VEL
LIN {X 0,Y 521.044,Z 978.19,A -85,B 0,C 180,E1 14723.836,E2 14723.836} C_VEL
LIN {X 0,Y 517.143,Z 998.663,A -85,B 0,C 180,E1 14723.036,E2 14723.036} C_VEL
LIN {X 0,Y 512.572,Z 1019.903,A -85,B 0,C 180,E1 14722.062,E2 14722.062} C_VEL
LIN {X 0,Y 506.301,Z 1046.044,A -85,B 0,C 180,E1 14720.631,E2 14720.631} C_VEL
LIN {X 0,Y 500.578,Z 1067.39,A -85,B 0,C 180,E1 14719.245,E2 14719.245} C_VEL
LIN {X 0,Y 495.312,Z 1085.76,A -85,B 0,C 180,E1 14717.883,E2 14717.883} C_VEL
LIN {X 0,Y 489.877,Z 1103.709,A -85,B 0,C 180,E1 14716.378,E2 14716.378} C_VEL
LIN {X 0,Y 484.018,Z 1122.306,A -85,B 0,C 180,E1 14714.61,E2 14714.61} C_VEL
LIN {X 0,Y 476.595,Z 1145.002,A -85,B 0,C 180,E1 14712.109,E2 14712.109} C_VEL
LIN {X 0,Y 471.073,Z 1161.427,A -85,B 0,C 180,E1 14710.02,E2 14710.02} C_VEL
LIN {X 0,Y 466.257,Z 1175.723,A -85,B 0,C 180,E1 14707.98,E2 14707.98} C_VEL
LIN {X 0,Y 461.673,Z 1189.497,A -85,B 0,C 180,E1 14705.78,E2 14705.78} C_VEL
LIN {X 0,Y 457.138,Z 1203.374,A -85,B 0,C 180,E1 14703.293,E2 14703.293} C_VEL
LIN {X 0,Y 451.981,Z 1219.996,A -85,B 0,C 180,E1 14699.846,E2 14699.846} C_VEL
LIN {X 0,Y 448.731,Z 1231.12,A -85,B 0,C 180,E1 14697.175,E2 14697.175} C_VEL
LIN {X 0,Y 446.138,Z 1240.969,A -85,B 0,C 180,E1 14694.49,E2 14694.49} C_VEL
LIN {X 0,Y 444.025,Z 1250.033,A -85,B 0,C 180,E1 14691.668,E2 14691.668} C_VEL
LIN {X 0,Y 442.115,Z 1259.619,A -85,B 0,C 180,E1 14688.181,E2 14688.181} C_VEL
LIN {X 0,Y 440.939,Z 1266.961,A -85,B 0,C 180,E1 14684.843,E2 14684.843} C_VEL
LIN {X 0,Y 440.395,Z 1271.982,A -85,B 0,C 180,E1 14682.052,E2 14682.052} C_VEL
LIN {X 0,Y 440.062,Z 1275.776,A -85,B 0,C 180,E1 14679.411,E2 14679.411} C_VEL
LIN {X 0,Y 439.963,Z 1278.74,A -85,B 0,C 180,E1 14676.652,E2 14676.652} C_VEL
LIN {X 0,Y 439.916,Z 1280.614,A -85,B 0,C 180,E1 14674.036,E2 14674.036} C_VEL
LIN {X 0,Y 439.9,Z 1281.571,A -85,B 0,C 180,E1 14671.429,E2 14671.429} C_VEL
LIN {X 0,Y 439.878,Z 1281.638,A -85,B 0,C 180,E1 14668.954,E2 14668.954} C_VEL
LIN {X 0,Y 439.916,Z 1280.815,A -85,B 0,C 180,E1 14666.348,E2 14666.348} C_VEL
LIN {X 0,Y 439.955,Z 1279.076,A -85,B 0,C 180,E1 14663.734,E2 14663.734} C_VEL
LIN {X 0,Y 440.054,Z 1276.25,A -85,B 0,C 180,E1 14660.977,E2 14660.977} C_VEL
LIN {X 0,Y 440.332,Z 1272.596,A -85,B 0,C 180,E1 14658.337,E2 14658.337} C_VEL
LIN {X 0,Y 440.813,Z 1267.973,A -85,B 0,C 180,E1 14655.682,E2 14655.682} C_VEL
LIN {X 0,Y 441.642,Z 1262.353,A -85,B 0,C 180,E1 14653.016,E2 14653.016} C_VEL
LIN {X 0,Y 442.882,Z 1255.343,A -85,B 0,C 180,E1 14650.202,E2 14650.202} C_VEL
LIN {X 0,Y 444.958,Z 1245.926,A -85,B 0,C 180,E1 14646.98,E2 14646.98} C_VEL
LIN {X 0,Y 447.914,Z 1234.207,A -85,B 0,C 180,E1 14643.623,E2 14643.623} C_VEL
LIN {X 0,Y 451.045,Z 1223.062,A -85,B 0,C 180,E1 14640.86,E2 14640.86} C_VEL
LIN {X 0,Y 454.628,Z 1211.296,A -85,B 0,C 180,E1 14638.286,E2 14638.286} C_VEL
LIN {X 0,Y 458.973,Z 1197.689,A -85,B 0,C 180,E1 14635.648,E2 14635.648} C_VEL
LIN {X 0,Y 465.142,Z 1179.058,A -85,B 0,C 180,E1 14632.527,E2 14632.527} C_VEL
LIN {X 0,Y 470.167,Z 1164.064,A -85,B 0,C 180,E1 14630.341,E2 14630.341} C_VEL
LIN {X 0,Y 475.335,Z 1148.639,A -85,B 0,C 180,E1 14628.337,E2 14628.337} C_VEL
LIN {X 0,Y 480.83,Z 1132.041,A -85,B 0,C 180,E1 14626.419,E2 14626.419} C_VEL
LIN {X 0,Y 487.806,Z 1110.56,A -85,B 0,C 180,E1 14624.24,E2 14624.24} C_VEL
LIN {X 0,Y 494.249,Z 1089.292,A -85,B 0,C 180,E1 14622.402,E2 14622.402} C_VEL
LIN {X 0,Y 499.544,Z 1070.933,A -85,B 0,C 180,E1 14621.007,E2 14621.007} C_VEL
LIN {X 0,Y 504.619,Z 1052.177,A -85,B 0,C 180,E1 14619.751,E2 14619.751} C_VEL
LIN {X 0,Y 509.685,Z 1032.059,A -85,B 0,C 180,E1 14618.576,E2 14618.576} C_VEL
LIN {X 0,Y 514.963,Z 1009.119,A -85,B 0,C 180,E1 14617.424,E2 14617.424} C_VEL
LIN {X 0,Y 520.148,Z 983.038,A -85,B 0,C 180,E1 14616.345,E2 14616.345} C_VEL
LIN {X 0,Y 523.972,Z 960.576,A -85,B 0,C 180,E1 14615.585,E2 14615.585} C_VEL
LIN {X 0,Y 527.047,Z 939.328,A -85,B 0,C 180,E1 14614.998,E2 14614.998} C_VEL
LIN {X 0,Y 529.644,Z 917.228,A -85,B 0,C 180,E1 14614.512,E2 14614.512} C_VEL
LIN {X 0,Y 531.899,Z 888.557,A -85,B 0,C 180,E1 14614.016,E2 14614.016} C_VEL
LIN {X 0,Y 543.99,Z 664.821,A -85,B 0,C 180,E1 14610.583,E2 14610.583} C_VEL
LIN {X 0,Y 549.586,Z 565.251,A -85,B 0,C 180,E1 14609.033,E2 14609.033} C_VEL
LIN {X 0,Y 538.454,Z 547.625,A -85,B 0,C 180,E1 14606.318,E2 14606.318} C_VEL
LIN {X 0,Y 529.923,Z 535.133,A -85,B 0,C 180,E1 14603.993,E2 14603.993} C_VEL
LIN {X 0,Y 522.853,Z 525.047,A -85,B 0,C 180,E1 14601.836,E2 14601.836} C_VEL
LIN {X 0,Y 517.963,Z 518.979,A -85,B 0,C 180,E1 14600.215,E2 14600.215} C_VEL
LIN {X 0,Y 513.876,Z 513.775,A -85,B 0,C 180,E1 14598.727,E2 14598.727} C_VEL
LIN {X 0,Y 509.832,Z 508.677,A -85,B 0,C 180,E1 14597.109,E2 14597.109} C_VEL
LIN {X 0,Y 506.252,Z 504.287,A -85,B 0,C 180,E1 14595.523,E2 14595.523} C_VEL
LIN {X 0,Y 505.092,Z 502.872,A -85,B 0,C 180,E1 14594.969,E2 14594.969} C_VEL
LIN {X 0,Y 501.557,Z 498.723,A -85,B 0,C 180,E1 14593.136,E2 14593.136} C_VEL
LIN {X 0,Y 500.613,Z 497.244,A -85,B 0,C 180,E1 14592.575,E2 14592.575} C_VEL
LIN {X 0,Y 497.418,Z 494.337,A -85,B 0,C 180,E1 14590.599,E2 14590.599} C_VEL
LIN {X 0,Y 495.647,Z 491.068,A -85,B 0,C 180,E1 14589.17,E2 14589.17} C_VEL
LIN {X 0,Y 491.878,Z 488.041,A -85,B 0,C 180,E1 14585.483,E2 14585.483} C_VEL
LIN {X 0,Y 490.592,Z 484.644,A -85,B 0,C 180,E1 14582.804,E2 14582.804} C_VEL
LIN {X 0,Y 490.744,Z 484.861,A -85,B 0,C 180,E1 14576.613,E2 14576.613} C_VEL
LIN {X 0,Y 492.166,Z 488.4,A -85,B 0,C 180,E1 14573.936,E2 14573.936} C_VEL
LIN {X 0,Y 495.825,Z 491.342,A -85,B 0,C 180,E1 14570.482,E2 14570.482} C_VEL
LIN {X 0,Y 498.045,Z 495.107,A -85,B 0,C 180,E1 14568.77,E2 14568.77} C_VEL
LIN {X 0,Y 501.06,Z 497.772,A -85,B 0,C 180,E1 14566.968,E2 14566.968} C_VEL
LIN {X 0,Y 504.124,Z 502.019,A -85,B 0,C 180,E1 14565.293,E2 14565.293} C_VEL
LIN {X 0,Y 505.989,Z 503.81,A -85,B 0,C 180,E1 14564.41,E2 14564.41} C_VEL
LIN {X 0,Y 509.653,Z 508.468,A -85,B 0,C 180,E1 14562.768,E2 14562.768} C_VEL
LIN {X 0,Y 511.099,Z 510.189,A -85,B 0,C 180,E1 14562.171,E2 14562.171} C_VEL
LIN {X 0,Y 515.764,Z 516.079,A -85,B 0,C 180,E1 14560.374,E2 14560.374} C_VEL
LIN {X 0,Y 520.544,Z 522.152,A -85,B 0,C 180,E1 14558.713,E2 14558.713} C_VEL
LIN {X 0,Y 525.013,Z 527.943,A -85,B 0,C 180,E1 14557.285,E2 14557.285} C_VEL
LIN {X 0,Y 531.722,Z 536.802,A -85,B 0,C 180,E1 14555.325,E2 14555.325} C_VEL
LIN {X 0,Y 541.17,Z 549.835,A -85,B 0,C 180,E1 14552.847,E2 14552.847} C_VEL
LIN {X 0,Y 548.728,Z 561.204,A -85,B 0,C 180,E1 14551.037,E2 14551.037} C_VEL
LIN {X 0,Y 549.647,Z 563.009,A -85,B 0,C 180,E1 14550.816,E2 14550.816} C_VEL
LIN {X 0,Y 537.251,Z 784.455,A -85,B 0,C 180,E1 14547.407,E2 14547.407} C_VEL
LIN {X 0,Y 531.094,Z 896.28,A -85,B 0,C 180,E1 14545.677,E2 14545.677} C_VEL
LIN {X 0,Y 528.457,Z 923.709,A -85,B 0,C 180,E1 14545.147,E2 14545.147} C_VEL
LIN {X 0,Y 524.818,Z 950.049,A -85,B 0,C 180,E1 14544.45,E2 14544.45} C_VEL
LIN {X 0,Y 521.338,Z 971.141,A -85,B 0,C 180,E1 14543.756,E2 14543.756} C_VEL
LIN {X 0,Y 517.44,Z 991.698,A -85,B 0,C 180,E1 14542.948,E2 14542.948} C_VEL
LIN {X 0,Y 512.88,Z 1012.984,A -85,B 0,C 180,E1 14541.965,E2 14541.965} C_VEL
LIN {X 0,Y 506.56,Z 1039.269,A -85,B 0,C 180,E1 14540.516,E2 14540.516} C_VEL
LIN {X 0,Y 500.793,Z 1060.7,A -85,B 0,C 180,E1 14539.113,E2 14539.113} C_VEL
LIN {X 0,Y 495.621,Z 1078.68,A -85,B 0,C 180,E1 14537.768,E2 14537.768} C_VEL
LIN {X 0,Y 490.325,Z 1096.085,A -85,B 0,C 180,E1 14536.299,E2 14536.299} C_VEL
LIN {X 0,Y 484.533,Z 1114.318,A -85,B 0,C 180,E1 14534.56,E2 14534.56} C_VEL
LIN {X 0,Y 477.207,Z 1136.546,A -85,B 0,C 180,E1 14532.107,E2 14532.107} C_VEL
LIN {X 0,Y 471.335,Z 1153.746,A -85,B 0,C 180,E1 14529.907,E2 14529.907} C_VEL
LIN {X 0,Y 466.394,Z 1168.21,A -85,B 0,C 180,E1 14527.82,E2 14527.82} C_VEL
LIN {X 0,Y 461.406,Z 1182.931,A -85,B 0,C 180,E1 14525.431,E2 14525.431} C_VEL
LIN {X 0,Y 455.972,Z 1199.484,A -85,B 0,C 180,E1 14522.351,E2 14522.351} C_VEL
LIN {X 0,Y 451.708,Z 1212.917,A -85,B 0,C 180,E1 14519.436,E2 14519.436} C_VEL
LIN {X 0,Y 448.659,Z 1223.22,A -85,B 0,C 180,E1 14516.901,E2 14516.901} C_VEL
LIN {X 0,Y 447.674,Z 1226.967,A -85,B 0,C 180,E1 14515.917,E2 14515.917} C_VEL
LIN {X 0,Y 445.852,Z 1230.328,A -85,B 0,C 180,E1 14515.05,E2 14515.05} C_VEL
LIN {X 0,Y 437.69,Z 1238.823,A -85,B 0,C 180,E1 14512.753,E2 14512.753} C_VEL
LIN {X 0,Y 436.373,Z 1241.271,A -85,B 0,C 180,E1 14511.959,E2 14511.959} C_VEL
LIN {X 0,Y 434.309,Z 1250.701,A -85,B 0,C 180,E1 14508.389,E2 14508.389} C_VEL
LIN {X 0,Y 433.09,Z 1257.626,A -85,B 0,C 180,E1 14505.126,E2 14505.126} C_VEL
LIN {X 0,Y 432.447,Z 1262.771,A -85,B 0,C 180,E1 14502.15,E2 14502.15} C_VEL
LIN {X 0,Y 432.085,Z 1266.46,A -85,B 0,C 180,E1 14499.46,E2 14499.46} C_VEL
LIN {X 0,Y 431.974,Z 1269.224,A -85,B 0,C 180,E1 14496.778,E2 14496.778} C_VEL
LIN {X 0,Y 431.919,Z 1271.072,A -85,B 0,C 180,E1 14494.119,E2 14494.119} C_VEL
LIN {X 0,Y 431.904,Z 1272.026,A -85,B 0,C 180,E1 14491.463,E2 14491.463} C_VEL
LIN {X 0,Y 431.884,Z 1272.088,A -85,B 0,C 180,E1 14488.81,E2 14488.81} C_VEL
LIN {X 0,Y 431.918,Z 1271.256,A -85,B 0,C 180,E1 14486.155,E2 14486.155} C_VEL
LIN {X 0,Y 431.967,Z 1269.528,A -85,B 0,C 180,E1 14483.492,E2 14483.492} C_VEL
LIN {X 0,Y 432.075,Z 1266.734,A -85,B 0,C 180,E1 14480.682,E2 14480.682} C_VEL
LIN {X 0,Y 432.408,Z 1263.124,A -85,B 0,C 180,E1 14477.993,E2 14477.993} C_VEL
LIN {X 0,Y 432.942,Z 1258.562,A -85,B 0,C 180,E1 14475.288,E2 14475.288} C_VEL
LIN {X 0,Y 433.868,Z 1253.016,A -85,B 0,C 180,E1 14472.571,E2 14472.571} C_VEL
LIN {X 0,Y 435.229,Z 1246.1,A -85,B 0,C 180,E1 14469.707,E2 14469.707} C_VEL
LIN {X 0,Y 437.603,Z 1236.399,A -85,B 0,C 180,E1 14466.293,E2 14466.293} C_VEL
LIN {X 0,Y 440.823,Z 1224.676,A -85,B 0,C 180,E1 14462.882,E2 14462.882} C_VEL
LIN {X 0,Y 444.129,Z 1213.958,A -85,B 0,C 180,E1 14460.168,E2 14460.168} C_VEL
LIN {X 0,Y 447.895,Z 1202.518,A -85,B 0,C 180,E1 14457.609,E2 14457.609} C_VEL
LIN {X 0,Y 452.785,Z 1188.267,A -85,B 0,C 180,E1 14454.793,E2 14454.793} C_VEL
LIN {X 0,Y 459.038,Z 1170.531,A -85,B 0,C 180,E1 14451.792,E2 14451.792} C_VEL
LIN {X 0,Y 464.468,Z 1155.26,A -85,B 0,C 180,E1 14449.536,E2 14449.536} C_VEL
LIN {X 0,Y 469.873,Z 1139.968,A -85,B 0,C 180,E1 14447.53,E2 14447.53} C_VEL
LIN {X 0,Y 475.824,Z 1122.878,A -85,B 0,C 180,E1 14445.544,E2 14445.544} C_VEL
LIN {X 0,Y 483.368,Z 1100.355,A -85,B 0,C 180,E1 14443.277,E2 14443.277} C_VEL
LIN {X 0,Y 489.513,Z 1080.896,A -85,B 0,C 180,E1 14441.595,E2 14441.595} C_VEL
LIN {X 0,Y 494.913,Z 1062.809,A -85,B 0,C 180,E1 14440.218,E2 14440.218} C_VEL
LIN {X 0,Y 500.145,Z 1044.04,A -85,B 0,C 180,E1 14438.959,E2 14438.959} C_VEL
LIN {X 0,Y 505.613,Z 1022.885,A -85,B 0,C 180,E1 14437.727,E2 14437.727} C_VEL
LIN {X 0,Y 511.808,Z 995.886,A -85,B 0,C 180,E1 14436.409,E2 14436.409} C_VEL
LIN {X 0,Y 516.119,Z 974.192,A -85,B 0,C 180,E1 14435.535,E2 14435.535} C_VEL
LIN {X 0,Y 519.785,Z 952.92,A -85,B 0,C 180,E1 14434.818,E2 14434.818} C_VEL
LIN {X 0,Y 522.91,Z 931.489,A -85,B 0,C 180,E1 14434.227,E2 14434.227} C_VEL
LIN {X 0,Y 525.676,Z 907.87,A -85,B 0,C 180,E1 14433.712,E2 14433.712} C_VEL
LIN {X 0,Y 528.227,Z 871.902,A -85,B 0,C 180,E1 14433.115,E2 14433.115} C_VEL
LIN {X 0,Y 540.635,Z 651.454,A -85,B 0,C 180,E1 14429.72,E2 14429.72} C_VEL
LIN {X 0,Y 545.515,Z 567.113,A -85,B 0,C 180,E1 14428.396,E2 14428.396} C_VEL
LIN {X 0,Y 538.403,Z 556.391,A -85,B 0,C 180,E1 14426.648,E2 14426.648} C_VEL
LIN {X 0,Y 528.439,Z 542.407,A -85,B 0,C 180,E1 14423.946,E2 14423.946} C_VEL
LIN {X 0,Y 520.397,Z 531.788,A -85,B 0,C 180,E1 14421.471,E2 14421.471} C_VEL
LIN {X 0,Y 516.233,Z 526.478,A -85,B 0,C 180,E1 14420.05,E2 14420.05} C_VEL
LIN {X 0,Y 512.217,Z 521.31,A -85,B 0,C 180,E1 14418.554,E2 14418.554} C_VEL
LIN {X 0,Y 508.25,Z 516.261,A -85,B 0,C 180,E1 14416.928,E2 14416.928} C_VEL
LIN {X 0,Y 504.642,Z 511.694,A -85,B 0,C 180,E1 14415.279,E2 14415.279} C_VEL
LIN {X 0,Y 500.086,Z 506.189,A -85,B 0,C 180,E1 14412.882,E2 14412.882} C_VEL
LIN {X 0,Y 499.249,Z 505,A -85,B 0,C 180,E1 14412.374,E2 14412.374} C_VEL
LIN {X 0,Y 496.088,Z 501.952,A -85,B 0,C 180,E1 14410.334,E2 14410.334} C_VEL
LIN {X 0,Y 494.454,Z 498.934,A -85,B 0,C 180,E1 14408.958,E2 14408.958} C_VEL
LIN {X 0,Y 490.735,Z 495.737,A -85,B 0,C 180,E1 14405.026,E2 14405.026} C_VEL
LIN {X 0,Y 489.703,Z 492.612,A -85,B 0,C 180,E1 14402.458,E2 14402.458} C_VEL
LIN {X 0,Y 489.766,Z 492.791,A -85,B 0,C 180,E1 14397.426,E2 14397.426} C_VEL
LIN {X 0,Y 491.65,Z 496.987,A -85,B 0,C 180,E1 14393.812,E2 14393.812} C_VEL
LIN {X 0,Y 494.716,Z 499.271,A -85,B 0,C 180,E1 14390.929,E2 14390.929} C_VEL
LIN {X 0,Y 497.03,Z 503.197,A -85,B 0,C 180,E1 14389.1,E2 14389.1} C_VEL
LIN {X 0,Y 499.802,Z 505.667,A -85,B 0,C 180,E1 14387.405,E2 14387.405} C_VEL
LIN {X 0,Y 503.141,Z 510.131,A -85,B 0,C 180,E1 14385.558,E2 14385.558} C_VEL
LIN {X 0,Y 504.62,Z 511.711,A -85,B 0,C 180,E1 14384.838,E2 14384.838} C_VEL
LIN {X 0,Y 508.228,Z 516.266,A -85,B 0,C 180,E1 14383.189,E2 14383.189} C_VEL
LIN {X 0,Y 513.952,Z 523.52,A -85,B 0,C 180,E1 14380.893,E2 14380.893} C_VEL
LIN {X 0,Y 518.793,Z 529.792,A -85,B 0,C 180,E1 14379.17,E2 14379.17} C_VEL
LIN {X 0,Y 523.279,Z 535.666,A -85,B 0,C 180,E1 14377.71,E2 14377.71} C_VEL
LIN {X 0,Y 531.78,Z 548.22,A -85,B 0,C 180,E1 14375.18,E2 14375.18} C_VEL
LIN {X 0,Y 539.424,Z 560.075,A -85,B 0,C 180,E1 14373.139,E2 14373.139} C_VEL
LIN {X 0,Y 545.567,Z 570.139,A -85,B 0,C 180,E1 14371.621,E2 14371.621} C_VEL
LIN {X 0,Y 533.125,Z 785.866,A -85,B 0,C 180,E1 14368.289,E2 14368.289} C_VEL
LIN {X 0,Y 526.508,Z 902.623,A -85,B 0,C 180,E1 14366.477,E2 14366.477} C_VEL
LIN {X 0,Y 523.791,Z 930.072,A -85,B 0,C 180,E1 14365.952,E2 14365.952} C_VEL
LIN {X 0,Y 520.034,Z 956.362,A -85,B 0,C 180,E1 14365.267,E2 14365.267} C_VEL
LIN {X 0,Y 516.443,Z 977.369,A -85,B 0,C 180,E1 14364.588,E2 14364.588} C_VEL
LIN {X 0,Y 512.523,Z 997.48,A -85,B 0,C 180,E1 14363.808,E2 14363.808} C_VEL
LIN {X 0,Y 508.189,Z 1017.212,A -85,B 0,C 180,E1 14362.916,E2 14362.916} C_VEL
LIN {X 0,Y 503.142,Z 1038.128,A -85,B 0,C 180,E1 14361.811,E2 14361.811} C_VEL
LIN {X 0,Y 496.29,Z 1063.695,A -85,B 0,C 180,E1 14360.221,E2 14360.221} C_VEL
LIN {X 0,Y 490.242,Z 1084.201,A -85,B 0,C 180,E1 14358.72,E2 14358.72} C_VEL
LIN {X 0,Y 484.509,Z 1102.565,A -85,B 0,C 180,E1 14357.185,E2 14357.185} C_VEL
LIN {X 0,Y 478.504,Z 1120.996,A -85,B 0,C 180,E1 14355.436,E2 14355.436} C_VEL
LIN {X 0,Y 471.436,Z 1142.038,A -85,B 0,C 180,E1 14353.146,E2 14353.146} C_VEL
LIN {X 0,Y 464.988,Z 1160.458,A -85,B 0,C 180,E1 14350.806,E2 14350.806} C_VEL
LIN {X 0,Y 459.654,Z 1175.633,A -85,B 0,C 180,E1 14348.625,E2 14348.625} C_VEL
LIN {X 0,Y 454.869,Z 1189.406,A -85,B 0,C 180,E1 14346.4,E2 14346.4} C_VEL
LIN {X 0,Y 450.131,Z 1203.283,A -85,B 0,C 180,E1 14343.88,E2 14343.88} C_VEL
LIN {X 0,Y 444.699,Z 1219.905,A -85,B 0,C 180,E1 14340.385,E2 14340.385} C_VEL
LIN {X 0,Y 441.226,Z 1231.242,A -85,B 0,C 180,E1 14337.616,E2 14337.616} C_VEL
LIN {X 0,Y 438.548,Z 1240.879,A -85,B 0,C 180,E1 14334.943,E2 14334.943} C_VEL
LIN {X 0,Y 436.301,Z 1249.942,A -85,B 0,C 180,E1 14332.071,E2 14332.071} C_VEL
LIN {X 0,Y 434.34,Z 1259.193,A -85,B 0,C 180,E1 14328.657,E2 14328.657} C_VEL
LIN {X 0,Y 433.024,Z 1266.871,A -85,B 0,C 180,E1 14325.12,E2 14325.12} C_VEL
LIN {X 0,Y 432.431,Z 1271.893,A -85,B 0,C 180,E1 14322.278,E2 14322.278} C_VEL
LIN {X 0,Y 432.077,Z 1275.688,A -85,B 0,C 180,E1 14319.587,E2 14319.587} C_VEL
LIN {X 0,Y 431.965,Z 1278.652,A -85,B 0,C 180,E1 14316.776,E2 14316.776} C_VEL
LIN {X 0,Y 431.917,Z 1280.526,A -85,B 0,C 180,E1 14314.111,E2 14314.111} C_VEL
LIN {X 0,Y 431.902,Z 1281.483,A -85,B 0,C 180,E1 14311.455,E2 14311.455} C_VEL
LIN {X 0,Y 431.879,Z 1281.55,A -85,B 0,C 180,E1 14308.935,E2 14308.935} C_VEL
LIN {X 0,Y 431.916,Z 1280.728,A -85,B 0,C 180,E1 14306.28,E2 14306.28} C_VEL
LIN {X 0,Y 431.959,Z 1278.988,A -85,B 0,C 180,E1 14303.617,E2 14303.617} C_VEL
LIN {X 0,Y 432.056,Z 1276.162,A -85,B 0,C 180,E1 14300.808,E2 14300.808} C_VEL
LIN {X 0,Y 432.368,Z 1272.507,A -85,B 0,C 180,E1 14298.119,E2 14298.119} C_VEL
LIN {X 0,Y 432.877,Z 1267.883,A -85,B 0,C 180,E1 14295.414,E2 14295.414} C_VEL
LIN {X 0,Y 433.771,Z 1262.263,A -85,B 0,C 180,E1 14292.698,E2 14292.698} C_VEL
LIN {X 0,Y 435.087,Z 1255.252,A -85,B 0,C 180,E1 14289.832,E2 14289.832} C_VEL
LIN {X 0,Y 437.182,Z 1246.243,A -85,B 0,C 180,E1 14286.689,E2 14286.689} C_VEL
LIN {X 0,Y 440.407,Z 1234.114,A -85,B 0,C 180,E1 14283.138,E2 14283.138} C_VEL
LIN {X 0,Y 443.613,Z 1223.337,A -85,B 0,C 180,E1 14280.419,E2 14280.419} C_VEL
LIN {X 0,Y 447.283,Z 1211.842,A -85,B 0,C 180,E1 14277.854,E2 14277.854} C_VEL
LIN {X 0,Y 451.549,Z 1199.005,A -85,B 0,C 180,E1 14275.311,E2 14275.311} C_VEL
LIN {X 0,Y 457.353,Z 1182.359,A -85,B 0,C 180,E1 14272.411,E2 14272.411} C_VEL
LIN {X 0,Y 463.435,Z 1164.838,A -85,B 0,C 180,E1 14269.799,E2 14269.799} C_VEL
LIN {X 0,Y 468.926,Z 1149.084,A -85,B 0,C 180,E1 14267.724,E2 14267.724} C_VEL
LIN {X 0,Y 474.433,Z 1133.061,A -85,B 0,C 180,E1 14265.847,E2 14265.847} C_VEL
LIN {X 0,Y 480.565,Z 1114.768,A -85,B 0,C 180,E1 14263.951,E2 14263.951} C_VEL
LIN {X 0,Y 488.263,Z 1090.672,A -85,B 0,C 180,E1 14261.803,E2 14261.803} C_VEL
LIN {X 0,Y 493.925,Z 1071.71,A -85,B 0,C 180,E1 14260.348,E2 14260.348} C_VEL
LIN {X 0,Y 499.227,Z 1052.751,A -85,B 0,C 180,E1 14259.069,E2 14259.069} C_VEL
LIN {X 0,Y 504.37,Z 1032.971,A -85,B 0,C 180,E1 14257.905,E2 14257.905} C_VEL
LIN {X 0,Y 509.258,Z 1012.422,A -85,B 0,C 180,E1 14256.859,E2 14256.859} C_VEL
LIN {X 0,Y 514.722,Z 986.647,A -85,B 0,C 180,E1 14255.754,E2 14255.754} C_VEL
LIN {X 0,Y 519.161,Z 961.434,A -85,B 0,C 180,E1 14254.889,E2 14254.889} C_VEL
LIN {X 0,Y 522.361,Z 940.011,A -85,B 0,C 180,E1 14254.294,E2 14254.294} C_VEL
LIN {X 0,Y 525.001,Z 918.308,A -85,B 0,C 180,E1 14253.813,E2 14253.813} C_VEL
LIN {X 0,Y 527.188,Z 892.55,A -85,B 0,C 180,E1 14253.359,E2 14253.359} C_VEL
LIN {X 0,Y 539.694,Z 668.938,A -85,B 0,C 180,E1 14249.913,E2 14249.913} C_VEL
LIN {X 0,Y 545.401,Z 569.81,A -85,B 0,C 180,E1 14248.358,E2 14248.358} C_VEL
LIN {X 0,Y 535.832,Z 554.373,A -85,B 0,C 180,E1 14245.95,E2 14245.95} C_VEL
LIN {X 0,Y 526.174,Z 539.867,A -85,B 0,C 180,E1 14243.223,E2 14243.223} C_VEL
LIN {X 0,Y 520.411,Z 531.858,A -85,B 0,C 180,E1 14241.411,E2 14241.411} C_VEL
LIN {X 0,Y 515.928,Z 526.172,A -85,B 0,C 180,E1 14239.885,E2 14239.885} C_VEL
LIN {X 0,Y 512.196,Z 521.32,A -85,B 0,C 180,E1 14238.495,E2 14238.495} C_VEL
LIN {X 0,Y 508.209,Z 516.246,A -85,B 0,C 180,E1 14236.87,E2 14236.87} C_VEL
LIN {X 0,Y 504.58,Z 511.65,A -85,B 0,C 180,E1 14235.222,E2 14235.222} C_VEL
LIN {X 0,Y 499.995,Z 506.105,A -85,B 0,C 180,E1 14232.825,E2 14232.825} C_VEL
LIN {X 0,Y 499.047,Z 504.884,A -85,B 0,C 180,E1 14232.262,E2 14232.262} C_VEL
LIN {X 0,Y 495.893,Z 501.679,A -85,B 0,C 180,E1 14230.221,E2 14230.221} C_VEL
LIN {X 0,Y 494.378,Z 498.9,A -85,B 0,C 180,E1 14228.959,E2 14228.959} C_VEL
LIN {X 0,Y 490.741,Z 495.784,A -85,B 0,C 180,E1 14225.261,E2 14225.261} C_VEL
LIN {X 0,Y 489.619,Z 492.584,A -85,B 0,C 180,E1 14222.809,E2 14222.809} C_VEL
LIN {X 0,Y 489.72,Z 492.756,A -85,B 0,C 180,E1 14216.723,E2 14216.723} C_VEL
LIN {X 0,Y 491.19,Z 496.398,A -85,B 0,C 180,E1 14213.924,E2 14213.924} C_VEL
LIN {X 0,Y 494.629,Z 499.2,A -85,B 0,C 180,E1 14210.635,E2 14210.635} C_VEL
LIN {X 0,Y 496.902,Z 503.001,A -85,B 0,C 180,E1 14208.862,E2 14208.862} C_VEL
LIN {X 0,Y 499.692,Z 505.492,A -85,B 0,C 180,E1 14207.167,E2 14207.167} C_VEL
LIN {X 0,Y 502.821,Z 509.822,A -85,B 0,C 180,E1 14205.43,E2 14205.43} C_VEL
LIN {X 0,Y 504.542,Z 511.551,A -85,B 0,C 180,E1 14204.6,E2 14204.6} C_VEL
LIN {X 0,Y 508.297,Z 516.278,A -85,B 0,C 180,E1 14202.897,E2 14202.897} C_VEL
LIN {X 0,Y 513.986,Z 523.546,A -85,B 0,C 180,E1 14200.629,E2 14200.629} C_VEL
LIN {X 0,Y 518.777,Z 529.73,A -85,B 0,C 180,E1 14198.933,E2 14198.933} C_VEL
LIN {X 0,Y 525.224,Z 538.079,A -85,B 0,C 180,E1 14196.881,E2 14196.881} C_VEL
LIN {X 0,Y 535.544,Z 552.33,A -85,B 0,C 180,E1 14193.975,E2 14193.975} C_VEL
LIN {X 0,Y 544.552,Z 565.62,A -85,B 0,C 180,E1 14191.723,E2 14191.723} C_VEL
LIN {X 0,Y 545.512,Z 567.559,A -85,B 0,C 180,E1 14191.483,E2 14191.483} C_VEL
LIN {X 0,Y 532.731,Z 788.891,A -85,B 0,C 180,E1 14188.067,E2 14188.067} C_VEL
LIN {X 0,Y 526.613,Z 896.391,A -85,B 0,C 180,E1 14186.398,E2 14186.398} C_VEL
LIN {X 0,Y 523.909,Z 923.813,A -85,B 0,C 180,E1 14185.868,E2 14185.868} C_VEL
LIN {X 0,Y 520.202,Z 950.009,A -85,B 0,C 180,E1 14185.175,E2 14185.175} C_VEL
LIN {X 0,Y 516.602,Z 971.239,A -85,B 0,C 180,E1 14184.479,E2 14184.479} C_VEL
LIN {X 0,Y 512.6,Z 991.796,A -85,B 0,C 180,E1 14183.671,E2 14183.671} C_VEL
LIN {X 0,Y 507.807,Z 1013.536,A -85,B 0,C 180,E1 14182.666,E2 14182.666} C_VEL
LIN {X 0,Y 501.182,Z 1040.173,A -85,B 0,C 180,E1 14181.187,E2 14181.187} C_VEL
LIN {X 0,Y 495.403,Z 1061.006,A -85,B 0,C 180,E1 14179.815,E2 14179.815} C_VEL
LIN {X 0,Y 490.045,Z 1079.028,A -85,B 0,C 180,E1 14178.461,E2 14178.461} C_VEL
LIN {X 0,Y 484.43,Z 1096.861,A -85,B 0,C 180,E1 14176.945,E2 14176.945} C_VEL
LIN {X 0,Y 477.977,Z 1116.513,A -85,B 0,C 180,E1 14175.044,E2 14175.044} C_VEL
LIN {X 0,Y 470.694,Z 1137.65,A -85,B 0,C 180,E1 14172.662,E2 14172.662} C_VEL
LIN {X 0,Y 465.154,Z 1153.306,A -85,B 0,C 180,E1 14170.641,E2 14170.641} C_VEL
LIN {X 0,Y 459.874,Z 1168.121,A -85,B 0,C 180,E1 14168.488,E2 14168.488} C_VEL
LIN {X 0,Y 454.747,Z 1182.642,A -85,B 0,C 180,E1 14166.108,E2 14166.108} C_VEL
LIN {X 0,Y 449.122,Z 1198.948,A -85,B 0,C 180,E1 14163.058,E2 14163.058} C_VEL
LIN {X 0,Y 444.479,Z 1212.901,A -85,B 0,C 180,E1 14159.992,E2 14159.992} C_VEL
LIN {X 0,Y 441.133,Z 1223.617,A -85,B 0,C 180,E1 14157.311,E2 14157.311} C_VEL
LIN {X 0,Y 438.374,Z 1233.375,A -85,B 0,C 180,E1 14154.53,E2 14154.53} C_VEL
LIN {X 0,Y 436.373,Z 1241.271,A -85,B 0,C 180,E1 14151.959,E2 14151.959} C_VEL
LIN {X 0,Y 434.765,Z 1244.109,A -85,B 0,C 180,E1 14151.03,E2 14151.03} C_VEL
LIN {X 0,Y 427.003,Z 1251.287,A -85,B 0,C 180,E1 14148.489,E2 14148.489} C_VEL
LIN {X 0,Y 426.033,Z 1253.01,A -85,B 0,C 180,E1 14147.713,E2 14147.713} C_VEL
LIN {X 0,Y 425.059,Z 1258.472,A -85,B 0,C 180,E1 14145,E2 14145} C_VEL
LIN {X 0,Y 424.469,Z 1263.066,A -85,B 0,C 180,E1 14142.243,E2 14142.243} C_VEL
LIN {X 0,Y 424.093,Z 1266.707,A -85,B 0,C 180,E1 14139.503,E2 14139.503} C_VEL
LIN {X 0,Y 423.976,Z 1269.421,A -85,B 0,C 180,E1 14136.776,E2 14136.776} C_VEL
LIN {X 0,Y 423.92,Z 1271.227,A -85,B 0,C 180,E1 14134.061,E2 14134.061} C_VEL
LIN {X 0,Y 423.9,Z 1272.136,A -85,B 0,C 180,E1 14131.355,E2 14131.355} C_VEL
LIN {X 0,Y 423.893,Z 1272.153,A -85,B 0,C 180,E1 14128.652,E2 14128.652} C_VEL
LIN {X 0,Y 423.921,Z 1271.276,A -85,B 0,C 180,E1 14125.946,E2 14125.946} C_VEL
LIN {X 0,Y 423.975,Z 1269.442,A -85,B 0,C 180,E1 14123.158,E2 14123.158} C_VEL
LIN {X 0,Y 424.096,Z 1266.664,A -85,B 0,C 180,E1 14120.368,E2 14120.368} C_VEL
LIN {X 0,Y 424.477,Z 1263.007,A -85,B 0,C 180,E1 14117.627,E2 14117.627} C_VEL
LIN {X 0,Y 425.072,Z 1258.398,A -85,B 0,C 180,E1 14114.869,E2 14114.869} C_VEL
LIN {X 0,Y 426.132,Z 1252.504,A -85,B 0,C 180,E1 14111.962,E2 14111.962} C_VEL
LIN {X 0,Y 428.129,Z 1243.72,A -85,B 0,C 180,E1 14108.351,E2 14108.351} C_VEL
LIN {X 0,Y 430.856,Z 1233.318,A -85,B 0,C 180,E1 14104.875,E2 14104.875} C_VEL
LIN {X 0,Y 433.716,Z 1223.743,A -85,B 0,C 180,E1 14102.101,E2 14102.101} C_VEL
LIN {X 0,Y 437.275,Z 1212.908,A -85,B 0,C 180,E1 14099.348,E2 14099.348} C_VEL
LIN {X 0,Y 442.204,Z 1198.823,A -85,B 0,C 180,E1 14096.21,E2 14096.21} C_VEL
LIN {X 0,Y 447.84,Z 1183.233,A -85,B 0,C 180,E1 14093.254,E2 14093.254} C_VEL
LIN {X 0,Y 453.1,Z 1168.938,A -85,B 0,C 180,E1 14090.873,E2 14090.873} C_VEL
LIN {X 0,Y 458.52,Z 1154.34,A -85,B 0,C 180,E1 14088.718,E2 14088.718} C_VEL
LIN {X 0,Y 464.199,Z 1138.882,A -85,B 0,C 180,E1 14086.689,E2 14086.689} C_VEL
LIN {X 0,Y 471.424,Z 1118.892,A -85,B 0,C 180,E1 14084.383,E2 14084.383} C_VEL
LIN {X 0,Y 478.587,Z 1097.78,A -85,B 0,C 180,E1 14082.311,E2 14082.311} C_VEL
LIN {X 0,Y 484.687,Z 1079.039,A -85,B 0,C 180,E1 14080.708,E2 14080.708} C_VEL
LIN {X 0,Y 490.141,Z 1061.275,A -85,B 0,C 180,E1 14079.37,E2 14079.37} C_VEL
LIN {X 0,Y 495.815,Z 1041.428,A -85,B 0,C 180,E1 14078.056,E2 14078.056} C_VEL
LIN {X 0,Y 502.764,Z 1014.509,A -85,B 0,C 180,E1 14076.547,E2 14076.547} C_VEL
LIN {X 0,Y 507.577,Z 993.401,A -85,B 0,C 180,E1 14075.562,E2 14075.562} C_VEL
LIN {X 0,Y 511.822,Z 972.328,A -85,B 0,C 180,E1 14074.727,E2 14074.727} C_VEL
LIN {X 0,Y 515.561,Z 950.975,A -85,B 0,C 180,E1 14074.022,E2 14074.022} C_VEL
LIN {X 0,Y 519.003,Z 927.436,A -85,B 0,C 180,E1 14073.39,E2 14073.39} C_VEL
LIN {X 0,Y 522.159,Z 898.101,A -85,B 0,C 180,E1 14072.802,E2 14072.802} C_VEL
LIN {X 0,Y 526.147,Z 831.934,A -85,B 0,C 180,E1 14071.763,E2 14071.763} C_VEL
LIN {X 0,Y 538.779,Z 616.982,A -85,B 0,C 180,E1 14068.439,E2 14068.439} C_VEL
LIN {X 0,Y 541.509,Z 571.796,A -85,B 0,C 180,E1 14067.731,E2 14067.731} C_VEL
LIN {X 0,Y 532.671,Z 558.685,A -85,B 0,C 180,E1 14065.459,E2 14065.459} C_VEL
LIN {X 0,Y 523.004,Z 545.102,A -85,B 0,C 180,E1 14062.658,E2 14062.658} C_VEL
LIN {X 0,Y 515.266,Z 534.859,A -85,B 0,C 180,E1 14060.089,E2 14060.089} C_VEL
LIN {X 0,Y 510.411,Z 528.704,A -85,B 0,C 180,E1 14058.267,E2 14058.267} C_VEL
LIN {X 0,Y 506.64,Z 523.829,A -85,B 0,C 180,E1 14056.688,E2 14056.688} C_VEL
LIN {X 0,Y 502.989,Z 519.057,A -85,B 0,C 180,E1 14054.977,E2 14054.977} C_VEL
LIN {X 0,Y 498.814,Z 514.048,A -85,B 0,C 180,E1 14052.738,E2 14052.738} C_VEL
LIN {X 0,Y 497.895,Z 512.758,A -85,B 0,C 180,E1 14052.173,E2 14052.173} C_VEL
LIN {X 0,Y 494.733,Z 509.527,A -85,B 0,C 180,E1 14050.068,E2 14050.068} C_VEL
LIN {X 0,Y 493.343,Z 506.829,A -85,B 0,C 180,E1 14048.861,E2 14048.861} C_VEL
LIN {X 0,Y 489.686,Z 503.616,A -85,B 0,C 180,E1 14044.92,E2 14044.92} C_VEL
LIN {X 0,Y 488.688,Z 500.548,A -85,B 0,C 180,E1 14042.345,E2 14042.345} C_VEL
LIN {X 0,Y 488.753,Z 500.679,A -85,B 0,C 180,E1 14037.538,E2 14037.538} C_VEL
LIN {X 0,Y 490.58,Z 504.869,A -85,B 0,C 180,E1 14033.916,E2 14033.916} C_VEL
LIN {X 0,Y 493.528,Z 507.118,A -85,B 0,C 180,E1 14031.084,E2 14031.084} C_VEL
LIN {X 0,Y 495.89,Z 511.088,A -85,B 0,C 180,E1 14029.192,E2 14029.192} C_VEL
LIN {X 0,Y 498.443,Z 513.376,A -85,B 0,C 180,E1 14027.605,E2 14027.605} C_VEL
LIN {X 0,Y 501.84,Z 517.932,A -85,B 0,C 180,E1 14025.696,E2 14025.696} C_VEL
LIN {X 0,Y 503.182,Z 519.443,A -85,B 0,C 180,E1 14025.029,E2 14025.029} C_VEL
LIN {X 0,Y 506.876,Z 524.074,A -85,B 0,C 180,E1 14023.32,E2 14023.32} C_VEL
LIN {X 0,Y 512.258,Z 531.089,A -85,B 0,C 180,E1 14021.123,E2 14021.123} C_VEL
LIN {X 0,Y 516.961,Z 537.26,A -85,B 0,C 180,E1 14019.419,E2 14019.419} C_VEL
LIN {X 0,Y 521.552,Z 543.365,A -85,B 0,C 180,E1 14017.899,E2 14017.899} C_VEL
LIN {X 0,Y 530.772,Z 557.268,A -85,B 0,C 180,E1 14015.129,E2 14015.129} C_VEL
LIN {X 0,Y 538.692,Z 569.872,A -85,B 0,C 180,E1 14013.01,E2 14013.01} C_VEL
LIN {X 0,Y 541.493,Z 574.894,A -85,B 0,C 180,E1 14012.295,E2 14012.295} C_VEL
LIN {X 0,Y 528.587,Z 791.976,A -85,B 0,C 180,E1 14008.935,E2 14008.935} C_VEL
LIN {X 0,Y 522.104,Z 902.662,A -85,B 0,C 180,E1 14007.211,E2 14007.211} C_VEL
LIN {X 0,Y 519.297,Z 930.243,A -85,B 0,C 180,E1 14006.682,E2 14006.682} C_VEL
LIN {X 0,Y 515.479,Z 956.283,A -85,B 0,C 180,E1 14006.004,E2 14006.004} C_VEL
LIN {X 0,Y 511.796,Z 977.289,A -85,B 0,C 180,E1 14005.326,E2 14005.326} C_VEL
LIN {X 0,Y 507.645,Z 997.977,A -85,B 0,C 180,E1 14004.524,E2 14004.524} C_VEL
LIN {X 0,Y 503.05,Z 1018.261,A -85,B 0,C 180,E1 14003.601,E2 14003.601} C_VEL
LIN {X 0,Y 496.985,Z 1042.616,A -85,B 0,C 180,E1 14002.293,E2 14002.293} C_VEL
LIN {X 0,Y 490.325,Z 1066.051,A -85,B 0,C 180,E1 14000.788,E2 14000.788} C_VEL
LIN {X 0,Y 484.589,Z 1084.851,A -85,B 0,C 180,E1 13999.396,E2 13999.396} C_VEL
LIN {X 0,Y 478.684,Z 1103.148,A -85,B 0,C 180,E1 13997.854,E2 13997.854} C_VEL
LIN {X 0,Y 472.485,Z 1121.525,A -85,B 0,C 180,E1 13996.094,E2 13996.094} C_VEL
LIN {X 0,Y 464.797,Z 1143.455,A -85,B 0,C 180,E1 13993.666,E2 13993.666} C_VEL
LIN {X 0,Y 458.339,Z 1161.248,A -85,B 0,C 180,E1 13991.37,E2 13991.37} C_VEL
LIN {X 0,Y 452.802,Z 1176.393,A -85,B 0,C 180,E1 13989.158,E2 13989.158} C_VEL
LIN {X 0,Y 447.569,Z 1190.866,A -85,B 0,C 180,E1 13986.772,E2 13986.772} C_VEL
LIN {X 0,Y 441.496,Z 1207.958,A -85,B 0,C 180,E1 13983.54,E2 13983.54} C_VEL
LIN {X 0,Y 437.063,Z 1220.998,A -85,B 0,C 180,E1 13980.661,E2 13980.661} C_VEL
LIN {X 0,Y 433.556,Z 1231.975,A -85,B 0,C 180,E1 13977.91,E2 13977.91} C_VEL
LIN {X 0,Y 430.717,Z 1241.736,A -85,B 0,C 180,E1 13975.127,E2 13975.127} C_VEL
LIN {X 0,Y 427.994,Z 1252.479,A -85,B 0,C 180,E1 13971.593,E2 13971.593} C_VEL
LIN {X 0,Y 426.065,Z 1261.274,A -85,B 0,C 180,E1 13968.041,E2 13968.041} C_VEL
LIN {X 0,Y 425.029,Z 1267.295,A -85,B 0,C 180,E1 13965.132,E2 13965.132} C_VEL
LIN {X 0,Y 424.447,Z 1272.013,A -85,B 0,C 180,E1 13962.374,E2 13962.374} C_VEL
LIN {X 0,Y 424.081,Z 1275.761,A -85,B 0,C 180,E1 13959.632,E2 13959.632} C_VEL
LIN {X 0,Y 423.967,Z 1278.624,A -85,B 0,C 180,E1 13956.832,E2 13956.832} C_VEL
LIN {X 0,Y 423.917,Z 1280.438,A -85,B 0,C 180,E1 13954.189,E2 13954.189} C_VEL
LIN {X 0,Y 423.903,Z 1281.396,A -85,B 0,C 180,E1 13951.483,E2 13951.483} C_VEL
LIN {X 0,Y 423.881,Z 1281.463,A -85,B 0,C 180,E1 13948.915,E2 13948.915} C_VEL
LIN {X 0,Y 423.917,Z 1280.64,A -85,B 0,C 180,E1 13946.21,E2 13946.21} C_VEL
LIN {X 0,Y 423.961,Z 1278.9,A -85,B 0,C 180,E1 13943.496,E2 13943.496} C_VEL
LIN {X 0,Y 424.058,Z 1276.234,A -85,B 0,C 180,E1 13940.77,E2 13940.77} C_VEL
LIN {X 0,Y 424.384,Z 1272.626,A -85,B 0,C 180,E1 13938.03,E2 13938.03} C_VEL
LIN {X 0,Y 424.916,Z 1268.049,A -85,B 0,C 180,E1 13935.273,E2 13935.273} C_VEL
LIN {X 0,Y 425.85,Z 1262.479,A -85,B 0,C 180,E1 13932.507,E2 13932.507} C_VEL
LIN {X 0,Y 427.151,Z 1255.874,A -85,B 0,C 180,E1 13929.727,E2 13929.727} C_VEL
LIN {X 0,Y 428.995,Z 1248.193,A -85,B 0,C 180,E1 13926.945,E2 13926.945} C_VEL
LIN {X 0,Y 431.666,Z 1238.452,A -85,B 0,C 180,E1 13923.886,E2 13923.886} C_VEL
LIN {X 0,Y 435.957,Z 1224.398,A -85,B 0,C 180,E1 13920.149,E2 13920.149} C_VEL
LIN {X 0,Y 439.962,Z 1212.388,A -85,B 0,C 180,E1 13917.407,E2 13917.407} C_VEL
LIN {X 0,Y 444.142,Z 1200.321,A -85,B 0,C 180,E1 13914.962,E2 13914.962} C_VEL
LIN {X 0,Y 448.959,Z 1186.928,A -85,B 0,C 180,E1 13912.552,E2 13912.552} C_VEL
LIN {X 0,Y 455.532,Z 1169.051,A -85,B 0,C 180,E1 13909.721,E2 13909.721} C_VEL
LIN {X 0,Y 462.227,Z 1150.487,A -85,B 0,C 180,E1 13907.213,E2 13907.213} C_VEL
LIN {X 0,Y 467.885,Z 1134.639,A -85,B 0,C 180,E1 13905.323,E2 13905.323} C_VEL
LIN {X 0,Y 473.759,Z 1117.727,A -85,B 0,C 180,E1 13903.531,E2 13903.531} C_VEL
LIN {X 0,Y 480.041,Z 1098.977,A -85,B 0,C 180,E1 13901.78,E2 13901.78} C_VEL
LIN {X 0,Y 487.926,Z 1073.998,A -85,B 0,C 180,E1 13899.781,E2 13899.781} C_VEL
LIN {X 0,Y 493.779,Z 1053.792,A -85,B 0,C 180,E1 13898.401,E2 13898.401} C_VEL
LIN {X 0,Y 499.054,Z 1034.16,A -85,B 0,C 180,E1 13897.235,E2 13897.235} C_VEL
LIN {X 0,Y 503.871,Z 1014.594,A -85,B 0,C 180,E1 13896.227,E2 13896.227} C_VEL
LIN {X 0,Y 508.485,Z 993.798,A -85,B 0,C 180,E1 13895.306,E2 13895.306} C_VEL
LIN {X 0,Y 513.685,Z 966.919,A -85,B 0,C 180,E1 13894.322,E2 13894.322} C_VEL
LIN {X 0,Y 517.578,Z 941.999,A -85,B 0,C 180,E1 13893.61,E2 13893.61} C_VEL
LIN {X 0,Y 520.355,Z 920.112,A -85,B 0,C 180,E1 13893.115,E2 13893.115} C_VEL
LIN {X 0,Y 522.433,Z 897.466,A -85,B 0,C 180,E1 13892.707,E2 13892.707} C_VEL
LIN {X 0,Y 535.111,Z 679.093,A -85,B 0,C 180,E1 13889.325,E2 13889.325} C_VEL
LIN {X 0,Y 541.334,Z 574.376,A -85,B 0,C 180,E1 13887.681,E2 13887.681} C_VEL
LIN {X 0,Y 532.766,Z 560.447,A -85,B 0,C 180,E1 13885.454,E2 13885.454} C_VEL
LIN {X 0,Y 523.905,Z 546.896,A -85,B 0,C 180,E1 13882.884,E2 13882.884} C_VEL
LIN {X 0,Y 518.475,Z 539.22,A -85,B 0,C 180,E1 13881.139,E2 13881.139} C_VEL
LIN {X 0,Y 513.91,Z 533.36,A -85,B 0,C 180,E1 13879.551,E2 13879.551} C_VEL
LIN {X 0,Y 510.385,Z 528.713,A -85,B 0,C 180,E1 13878.209,E2 13878.209} C_VEL
LIN {X 0,Y 506.466,Z 523.69,A -85,B 0,C 180,E1 13876.576,E2 13876.576} C_VEL
LIN {X 0,Y 502.356,Z 518.377,A -85,B 0,C 180,E1 13874.642,E2 13874.642} C_VEL
LIN {X 0,Y 498.72,Z 513.965,A -85,B 0,C 180,E1 13872.682,E2 13872.682} C_VEL
LIN {X 0,Y 497.888,Z 512.762,A -85,B 0,C 180,E1 13872.173,E2 13872.173} C_VEL
LIN {X 0,Y 494.683,Z 509.486,A -85,B 0,C 180,E1 13870.069,E2 13870.069} C_VEL
LIN {X 0,Y 493.264,Z 506.793,A -85,B 0,C 180,E1 13868.862,E2 13868.862} C_VEL
LIN {X 0,Y 489.612,Z 503.522,A -85,B 0,C 180,E1 13865.038,E2 13865.038} C_VEL
LIN {X 0,Y 488.596,Z 500.518,A -85,B 0,C 180,E1 13862.698,E2 13862.698} C_VEL
LIN {X 0,Y 488.698,Z 500.652,A -85,B 0,C 180,E1 13856.832,E2 13856.832} C_VEL
LIN {X 0,Y 490.124,Z 504.277,A -85,B 0,C 180,E1 13854.028,E2 13854.028} C_VEL
LIN {X 0,Y 493.5,Z 507.202,A -85,B 0,C 180,E1 13850.731,E2 13850.731} C_VEL
LIN {X 0,Y 495.929,Z 511.077,A -85,B 0,C 180,E1 13848.84,E2 13848.84} C_VEL
LIN {X 0,Y 498.419,Z 513.379,A -85,B 0,C 180,E1 13847.31,E2 13847.31} C_VEL
LIN {X 0,Y 501.632,Z 517.731,A -85,B 0,C 180,E1 13845.513,E2 13845.513} C_VEL
LIN {X 0,Y 503.211,Z 519.468,A -85,B 0,C 180,E1 13844.735,E2 13844.735} C_VEL
LIN {X 0,Y 507.074,Z 524.205,A -85,B 0,C 180,E1 13842.973,E2 13842.973} C_VEL
LIN {X 0,Y 512.414,Z 531.301,A -85,B 0,C 180,E1 13840.81,E2 13840.81} C_VEL
LIN {X 0,Y 517.096,Z 537.407,A -85,B 0,C 180,E1 13839.128,E2 13839.128} C_VEL
LIN {X 0,Y 523.221,Z 545.478,A -85,B 0,C 180,E1 13837.144,E2 13837.144} C_VEL
LIN {X 0,Y 533.138,Z 559.353,A -85,B 0,C 180,E1 13834.297,E2 13834.297} C_VEL
LIN {X 0,Y 541.468,Z 571.776,A -85,B 0,C 180,E1 13832.166,E2 13832.166} C_VEL
LIN {X 0,Y 528.392,Z 791.424,A -85,B 0,C 180,E1 13828.768,E2 13828.768} C_VEL
LIN {X 0,Y 522.209,Z 896.61,A -85,B 0,C 180,E1 13827.129,E2 13827.129} C_VEL
LIN {X 0,Y 519.423,Z 924.084,A -85,B 0,C 180,E1 13826.597,E2 13826.597} C_VEL
LIN {X 0,Y 515.64,Z 950.154,A -85,B 0,C 180,E1 13825.908,E2 13825.908} C_VEL
LIN {X 0,Y 511.951,Z 971.337,A -85,B 0,C 180,E1 13825.215,E2 13825.215} C_VEL
LIN {X 0,Y 507.844,Z 991.893,A -85,B 0,C 180,E1 13824.407,E2 13824.407} C_VEL
LIN {X 0,Y 503.023,Z 1013.178,A -85,B 0,C 180,E1 13823.425,E2 13823.425} C_VEL
LIN {X 0,Y 496.34,Z 1039.461,A -85,B 0,C 180,E1 13821.971,E2 13821.971} C_VEL
LIN {X 0,Y 490.396,Z 1060.293,A -85,B 0,C 180,E1 13820.604,E2 13820.604} C_VEL
LIN {X 0,Y 484.928,Z 1078.139,A -85,B 0,C 180,E1 13819.269,E2 13819.269} C_VEL
LIN {X 0,Y 479.035,Z 1096.291,A -85,B 0,C 180,E1 13817.729,E2 13817.729} C_VEL
LIN {X 0,Y 472.844,Z 1114.509,A -85,B 0,C 180,E1 13815.972,E2 13815.972} C_VEL
LIN {X 0,Y 464.973,Z 1136.736,A -85,B 0,C 180,E1 13813.485,E2 13813.485} C_VEL
LIN {X 0,Y 458.856,Z 1153.383,A -85,B 0,C 180,E1 13811.322,E2 13811.322} C_VEL
LIN {X 0,Y 453.596,Z 1167.559,A -85,B 0,C 180,E1 13809.248,E2 13809.248} C_VEL
LIN {X 0,Y 448.285,Z 1181.971,A -85,B 0,C 180,E1 13806.872,E2 13806.872} C_VEL
LIN {X 0,Y 442.596,Z 1197.728,A -85,B 0,C 180,E1 13803.921,E2 13803.921} C_VEL
LIN {X 0,Y 437.399,Z 1212.536,A -85,B 0,C 180,E1 13800.652,E2 13800.652} C_VEL
LIN {X 0,Y 433.824,Z 1223.407,A -85,B 0,C 180,E1 13797.9,E2 13797.9} C_VEL
LIN {X 0,Y 430.941,Z 1233.013,A -85,B 0,C 180,E1 13795.129,E2 13795.129} C_VEL
LIN {X 0,Y 428.282,Z 1243.041,A -85,B 0,C 180,E1 13791.793,E2 13791.793} C_VEL
LIN {X 0,Y 426.169,Z 1252.294,A -85,B 0,C 180,E1 13788.044,E2 13788.044} C_VEL
LIN {X 0,Y 426.033,Z 1253.01,A -85,B 0,C 180,E1 13787.713,E2 13787.713} C_VEL
LIN {X 0,Y 424.674,Z 1255.252,A -85,B 0,C 180,E1 13786.728,E2 13786.728} C_VEL
LIN {X 0,Y 417.376,Z 1260.939,A -85,B 0,C 180,E1 13783.953,E2 13783.953} C_VEL
LIN {X 0,Y 416.656,Z 1262.093,A -85,B 0,C 180,E1 13783.211,E2 13783.211} C_VEL
LIN {X 0,Y 416.163,Z 1266.323,A -85,B 0,C 180,E1 13780.105,E2 13780.105} C_VEL
LIN {X 0,Y 415.995,Z 1269.285,A -85,B 0,C 180,E1 13777.184,E2 13777.184} C_VEL
LIN {X 0,Y 415.922,Z 1271.181,A -85,B 0,C 180,E1 13774.416,E2 13774.416} C_VEL
LIN {X 0,Y 415.907,Z 1272.179,A -85,B 0,C 180,E1 13771.657,E2 13771.657} C_VEL
LIN {X 0,Y 415.881,Z 1272.285,A -85,B 0,C 180,E1 13768.902,E2 13768.902} C_VEL
LIN {X 0,Y 415.92,Z 1271.476,A -85,B 0,C 180,E1 13766.099,E2 13766.099} C_VEL
LIN {X 0,Y 415.976,Z 1269.703,A -85,B 0,C 180,E1 13763.24,E2 13763.24} C_VEL
LIN {X 0,Y 416.095,Z 1267.067,A -85,B 0,C 180,E1 13760.46,E2 13760.46} C_VEL
LIN {X 0,Y 416.478,Z 1263.504,A -85,B 0,C 180,E1 13757.667,E2 13757.667} C_VEL
LIN {X 0,Y 417.085,Z 1258.99,A -85,B 0,C 180,E1 13754.857,E2 13754.857} C_VEL
LIN {X 0,Y 418.117,Z 1253.493,A -85,B 0,C 180,E1 13752.037,E2 13752.037} C_VEL
LIN {X 0,Y 419.562,Z 1246.977,A -85,B 0,C 180,E1 13749.206,E2 13749.206} C_VEL
LIN {X 0,Y 421.566,Z 1239.39,A -85,B 0,C 180,E1 13746.375,E2 13746.375} C_VEL
LIN {X 0,Y 424.917,Z 1228.4,A -85,B 0,C 180,E1 13742.844,E2 13742.844} C_VEL
LIN {X 0,Y 429.086,Z 1215.844,A -85,B 0,C 180,E1 13739.475,E2 13739.475} C_VEL
LIN {X 0,Y 433.348,Z 1203.958,A -85,B 0,C 180,E1 13736.698,E2 13736.698} C_VEL
LIN {X 0,Y 437.952,Z 1191.593,A -85,B 0,C 180,E1 13734.145,E2 13734.145} C_VEL
LIN {X 0,Y 444.125,Z 1175.661,A -85,B 0,C 180,E1 13731.26,E2 13731.26} C_VEL
LIN {X 0,Y 451.142,Z 1157.387,A -85,B 0,C 180,E1 13728.437,E2 13728.437} C_VEL
LIN {X 0,Y 457.015,Z 1141.995,A -85,B 0,C 180,E1 13726.356,E2 13726.356} C_VEL
LIN {X 0,Y 462.935,Z 1126.18,A -85,B 0,C 180,E1 13724.459,E2 13724.459} C_VEL
LIN {X 0,Y 469.058,Z 1109.289,A -85,B 0,C 180,E1 13722.664,E2 13722.664} C_VEL
LIN {X 0,Y 476.781,Z 1087.179,A -85,B 0,C 180,E1 13720.617,E2 13720.617} C_VEL
LIN {X 0,Y 483.755,Z 1065.336,A -85,B 0,C 180,E1 13718.905,E2 13718.905} C_VEL
LIN {X 0,Y 489.513,Z 1046.002,A -85,B 0,C 180,E1 13717.586,E2 13717.586} C_VEL
LIN {X 0,Y 495.005,Z 1026.057,A -85,B 0,C 180,E1 13716.404,E2 13716.404} C_VEL
LIN {X 0,Y 500.453,Z 1004.327,A -85,B 0,C 180,E1 13715.297,E2 13715.297} C_VEL
LIN {X 0,Y 506.424,Z 976.837,A -85,B 0,C 180,E1 13714.139,E2 13714.139} C_VEL
LIN {X 0,Y 510.545,Z 954.33,A -85,B 0,C 180,E1 13713.372,E2 13713.372} C_VEL
LIN {X 0,Y 513.819,Z 933.186,A -85,B 0,C 180,E1 13712.784,E2 13712.784} C_VEL
LIN {X 0,Y 516.545,Z 911.438,A -85,B 0,C 180,E1 13712.3,E2 13712.3} C_VEL
LIN {X 0,Y 518.95,Z 883.846,A -85,B 0,C 180,E1 13711.815,E2 13711.815} C_VEL
LIN {X 0,Y 532.15,Z 662.939,A -85,B 0,C 180,E1 13708.396,E2 13708.396} C_VEL
LIN {X 0,Y 537.558,Z 576.451,A -85,B 0,C 180,E1 13707.051,E2 13707.051} C_VEL
LIN {X 0,Y 527.508,Z 561.643,A -85,B 0,C 180,E1 13704.348,E2 13704.348} C_VEL
LIN {X 0,Y 519.379,Z 550.392,A -85,B 0,C 180,E1 13701.871,E2 13701.871} C_VEL
LIN {X 0,Y 513.244,Z 542.074,A -85,B 0,C 180,E1 13699.756,E2 13699.756} C_VEL
LIN {X 0,Y 508.482,Z 535.941,A -85,B 0,C 180,E1 13697.923,E2 13697.923} C_VEL
LIN {X 0,Y 505.039,Z 531.395,A -85,B 0,C 180,E1 13696.446,E2 13696.446} C_VEL
LIN {X 0,Y 500.895,Z 526.036,A -85,B 0,C 180,E1 13694.45,E2 13694.45} C_VEL
LIN {X 0,Y 497.278,Z 521.434,A -85,B 0,C 180,E1 13692.424,E2 13692.424} C_VEL
LIN {X 0,Y 496.171,Z 520.242,A -85,B 0,C 180,E1 13691.744,E2 13691.744} C_VEL
LIN {X 0,Y 493.18,Z 516.734,A -85,B 0,C 180,E1 13689.629,E2 13689.629} C_VEL
LIN {X 0,Y 492.09,Z 514.661,A -85,B 0,C 180,E1 13688.648,E2 13688.648} C_VEL
LIN {X 0,Y 488.51,Z 511.218,A -85,B 0,C 180,E1 13684.579,E2 13684.579} C_VEL
LIN {X 0,Y 487.676,Z 508.483,A -85,B 0,C 180,E1 13682.233,E2 13682.233} C_VEL
LIN {X 0,Y 487.765,Z 508.738,A -85,B 0,C 180,E1 13677.533,E2 13677.533} C_VEL
LIN {X 0,Y 489.606,Z 512.844,A -85,B 0,C 180,E1 13673.904,E2 13673.904} C_VEL
LIN {X 0,Y 492.345,Z 514.961,A -85,B 0,C 180,E1 13671.239,E2 13671.239} C_VEL
LIN {X 0,Y 494.75,Z 518.979,A -85,B 0,C 180,E1 13669.284,E2 13669.284} C_VEL
LIN {X 0,Y 497.178,Z 521.243,A -85,B 0,C 180,E1 13667.75,E2 13667.75} C_VEL
LIN {X 0,Y 500.652,Z 525.834,A -85,B 0,C 180,E1 13665.78,E2 13665.78} C_VEL
LIN {X 0,Y 501.964,Z 527.526,A -85,B 0,C 180,E1 13665.11,E2 13665.11} C_VEL
LIN {X 0,Y 506.388,Z 533.163,A -85,B 0,C 180,E1 13663.067,E2 13663.067} C_VEL
LIN {X 0,Y 510.709,Z 538.857,A -85,B 0,C 180,E1 13661.301,E2 13661.301} C_VEL
LIN {X 0,Y 515.364,Z 545.036,A -85,B 0,C 180,E1 13659.589,E2 13659.589} C_VEL
LIN {X 0,Y 519.585,Z 550.761,A -85,B 0,C 180,E1 13658.168,E2 13658.168} C_VEL
LIN {X 0,Y 528.418,Z 564.291,A -85,B 0,C 180,E1 13655.459,E2 13655.459} C_VEL
LIN {X 0,Y 536.129,Z 576.762,A -85,B 0,C 180,E1 13653.35,E2 13653.35} C_VEL
LIN {X 0,Y 537.52,Z 579.224,A -85,B 0,C 180,E1 13652.986,E2 13652.986} C_VEL
LIN {X 0,Y 524.179,Z 797.027,A -85,B 0,C 180,E1 13649.608,E2 13649.608} C_VEL
LIN {X 0,Y 517.789,Z 902.701,A -85,B 0,C 180,E1 13647.956,E2 13647.956} C_VEL
LIN {X 0,Y 514.899,Z 930.327,A -85,B 0,C 180,E1 13647.426,E2 13647.426} C_VEL
LIN {X 0,Y 510.992,Z 956.312,A -85,B 0,C 180,E1 13646.751,E2 13646.751} C_VEL
LIN {X 0,Y 507.238,Z 977.208,A -85,B 0,C 180,E1 13646.078,E2 13646.078} C_VEL
LIN {X 0,Y 502.973,Z 997.895,A -85,B 0,C 180,E1 13645.278,E2 13645.278} C_VEL
LIN {X 0,Y 498.257,Z 1018.178,A -85,B 0,C 180,E1 13644.355,E2 13644.355} C_VEL
LIN {X 0,Y 492.125,Z 1042.089,A -85,B 0,C 180,E1 13643.074,E2 13643.074} C_VEL
LIN {X 0,Y 485.157,Z 1065.965,A -85,B 0,C 180,E1 13641.542,E2 13641.542} C_VEL
LIN {X 0,Y 479.245,Z 1084.765,A -85,B 0,C 180,E1 13640.147,E2 13640.147} C_VEL
LIN {X 0,Y 472.949,Z 1103.664,A -85,B 0,C 180,E1 13638.545,E2 13638.545} C_VEL
LIN {X 0,Y 466.113,Z 1123.263,A -85,B 0,C 180,E1 13636.645,E2 13636.645} C_VEL
LIN {X 0,Y 458.115,Z 1145.089,A -85,B 0,C 180,E1 13634.173,E2 13634.173} C_VEL
LIN {X 0,Y 452.062,Z 1161.159,A -85,B 0,C 180,E1 13632.074,E2 13632.074} C_VEL
LIN {X 0,Y 446.309,Z 1176.303,A -85,B 0,C 180,E1 13629.84,E2 13629.84} C_VEL
LIN {X 0,Y 440.848,Z 1190.776,A -85,B 0,C 180,E1 13627.428,E2 13627.428} C_VEL
LIN {X 0,Y 434.505,Z 1207.867,A -85,B 0,C 180,E1 13624.153,E2 13624.153} C_VEL
LIN {X 0,Y 429.843,Z 1220.878,A -85,B 0,C 180,E1 13621.241,E2 13621.241} C_VEL
LIN {X 0,Y 426.167,Z 1231.884,A -85,B 0,C 180,E1 13618.437,E2 13618.437} C_VEL
LIN {X 0,Y 423.172,Z 1241.622,A -85,B 0,C 180,E1 13615.614,E2 13615.614} C_VEL
LIN {X 0,Y 420.32,Z 1252.211,A -85,B 0,C 180,E1 13612.072,E2 13612.072} C_VEL
LIN {X 0,Y 418.217,Z 1261.184,A -85,B 0,C 180,E1 13608.391,E2 13608.391} C_VEL
LIN {X 0,Y 417.126,Z 1267.205,A -85,B 0,C 180,E1 13605.426,E2 13605.426} C_VEL
LIN {X 0,Y 416.485,Z 1271.923,A -85,B 0,C 180,E1 13602.615,E2 13602.615} C_VEL
LIN {X 0,Y 416.097,Z 1275.672,A -85,B 0,C 180,E1 13599.819,E2 13599.819} C_VEL
LIN {X 0,Y 415.973,Z 1278.475,A -85,B 0,C 180,E1 13597.037,E2 13597.037} C_VEL
LIN {X 0,Y 415.918,Z 1280.35,A -85,B 0,C 180,E1 13594.27,E2 13594.27} C_VEL
LIN {X 0,Y 415.903,Z 1281.308,A -85,B 0,C 180,E1 13591.511,E2 13591.511} C_VEL
LIN {X 0,Y 415.882,Z 1281.375,A -85,B 0,C 180,E1 13588.894,E2 13588.894} C_VEL
LIN {X 0,Y 415.917,Z 1280.537,A -85,B 0,C 180,E1 13586.105,E2 13586.105} C_VEL
LIN {X 0,Y 415.963,Z 1278.812,A -85,B 0,C 180,E1 13583.371,E2 13583.371} C_VEL
LIN {X 0,Y 416.066,Z 1276.146,A -85,B 0,C 180,E1 13580.591,E2 13580.591} C_VEL
LIN {X 0,Y 416.428,Z 1272.476,A -85,B 0,C 180,E1 13577.757,E2 13577.757} C_VEL
LIN {X 0,Y 416.994,Z 1267.961,A -85,B 0,C 180,E1 13574.988,E2 13574.988} C_VEL
LIN {X 0,Y 417.986,Z 1262.388,A -85,B 0,C 180,E1 13572.167,E2 13572.167} C_VEL
LIN {X 0,Y 419.38,Z 1255.783,A -85,B 0,C 180,E1 13569.334,E2 13569.334} C_VEL
LIN {X 0,Y 421.331,Z 1248.1,A -85,B 0,C 180,E1 13566.5,E2 13566.5} C_VEL
LIN {X 0,Y 424.161,Z 1238.359,A -85,B 0,C 180,E1 13563.388,E2 13563.388} C_VEL
LIN {X 0,Y 428.694,Z 1224.305,A -85,B 0,C 180,E1 13559.591,E2 13559.591} C_VEL
LIN {X 0,Y 432.884,Z 1212.294,A -85,B 0,C 180,E1 13556.806,E2 13556.806} C_VEL
LIN {X 0,Y 437.524,Z 1199.522,A -85,B 0,C 180,E1 13554.191,E2 13554.191} C_VEL
LIN {X 0,Y 443.207,Z 1184.509,A -85,B 0,C 180,E1 13551.487,E2 13551.487} C_VEL
LIN {X 0,Y 450.454,Z 1165.429,A -85,B 0,C 180,E1 13548.531,E2 13548.531} C_VEL
LIN {X 0,Y 456.495,Z 1149.375,A -85,B 0,C 180,E1 13546.37,E2 13546.37} C_VEL
LIN {X 0,Y 462.358,Z 1133.537,A -85,B 0,C 180,E1 13544.482,E2 13544.482} C_VEL
LIN {X 0,Y 468.42,Z 1116.662,A -85,B 0,C 180,E1 13542.696,E2 13542.696} C_VEL
LIN {X 0,Y 475.751,Z 1095.532,A -85,B 0,C 180,E1 13540.739,E2 13540.739} C_VEL
LIN {X 0,Y 483.19,Z 1072.276,A -85,B 0,C 180,E1 13538.913,E2 13538.913} C_VEL
LIN {X 0,Y 488.983,Z 1052.795,A -85,B 0,C 180,E1 13537.59,E2 13537.59} C_VEL
LIN {X 0,Y 494.218,Z 1033.788,A -85,B 0,C 180,E1 13536.464,E2 13536.464} C_VEL
LIN {X 0,Y 499.1,Z 1014.497,A -85,B 0,C 180,E1 13535.473,E2 13535.473} C_VEL
LIN {X 0,Y 503.836,Z 993.702,A -85,B 0,C 180,E1 13534.553,E2 13534.553} C_VEL
LIN {X 0,Y 509.188,Z 966.713,A -85,B 0,C 180,E1 13533.567,E2 13533.567} C_VEL
LIN {X 0,Y 513.161,Z 941.899,A -85,B 0,C 180,E1 13532.86,E2 13532.86} C_VEL
LIN {X 0,Y 516.007,Z 920.009,A -85,B 0,C 180,E1 13532.368,E2 13532.368} C_VEL
LIN {X 0,Y 518.133,Z 897.359,A -85,B 0,C 180,E1 13531.959,E2 13531.959} C_VEL
LIN {X 0,Y 531.215,Z 678.981,A -85,B 0,C 180,E1 13528.568,E2 13528.568} C_VEL
